QRS_NEXT_CUT()
PTP {E1 28976.891,E2 28976.891}
PTP {X 0,Y 607.92,A -85,B 0,C 180,E1 28976.891,E2 28976.891,E3 0,E4 0,E5 0,E6 0}
QRS_SPEED_INIT()
LIN {X 0,Y 607.92,Z 1028,A -85,B 0,C 180,E1 28976.891,E2 28976.891,E3 0,E4 0,E5 0,E6 0} C_VEL
LIN {X 0,Y 607.92,Z 449.836,A -85,B 0,C 180,E1 28976.891,E2 28976.891} C_VEL
LIN {X 0,Y 607.92,Z 441.762,A -85,B 0,C 180,E1 28976.891,E2 28976.891} C_VEL
LIN {X 0,Y 607.916,Z 439.762,A -85,B 0,C 180,E1 28976.702,E2 28976.702} C_VEL
LIN {X 0,Y 607.879,Z 439.765,A -85,B 0,C 180,E1 28973.483,E2 28973.483} C_VEL
LIN {X 0,Y 607.903,Z 439.761,A -85,B 0,C 180,E1 28970.246,E2 28970.246} C_VEL
LIN {X 0,Y 607.86,Z 439.764,A -85,B 0,C 180,E1 28967.266,E2 28967.266} C_VEL
LIN {X 0,Y 607.883,Z 439.762,A -85,B 0,C 180,E1 28963.959,E2 28963.959} C_VEL
LIN {X 0,Y 607.887,Z 439.761,A -85,B 0,C 180,E1 28960.894,E2 28960.894} C_VEL
LIN {X 0,Y 607.863,Z 439.765,A -85,B 0,C 180,E1 28957.668,E2 28957.668} C_VEL
LIN {X 0,Y 607.909,Z 439.763,A -85,B 0,C 180,E1 28954.682,E2 28954.682} C_VEL
LIN {X 0,Y 607.904,Z 439.766,A -85,B 0,C 180,E1 28951.511,E2 28951.511} C_VEL
LIN {X 0,Y 607.907,Z 439.765,A -85,B 0,C 180,E1 28948.353,E2 28948.353} C_VEL
LIN {X 0,Y 607.906,Z 439.763,A -85,B 0,C 180,E1 28945.158,E2 28945.158} C_VEL
LIN {X 0,Y 607.884,Z 439.763,A -85,B 0,C 180,E1 28942.036,E2 28942.036} C_VEL
LIN {X 0,Y 607.88,Z 439.763,A -85,B 0,C 180,E1 28938.857,E2 28938.857} C_VEL
LIN {X 0,Y 607.897,Z 439.76,A -85,B 0,C 180,E1 28935.782,E2 28935.782} C_VEL
LIN {X 0,Y 607.855,Z 439.765,A -85,B 0,C 180,E1 28932.535,E2 28932.535} C_VEL
LIN {X 0,Y 607.91,Z 439.76,A -85,B 0,C 180,E1 28929.521,E2 28929.521} C_VEL
LIN {X 0,Y 607.877,Z 439.765,A -85,B 0,C 180,E1 28926.296,E2 28926.296} C_VEL
LIN {X 0,Y 607.914,Z 439.762,A -85,B 0,C 180,E1 28923.096,E2 28923.096} C_VEL
LIN {X 0,Y 607.914,Z 439.902,A -85,B 0,C 180,E1 28921.609,E2 28921.609} C_VEL
LIN {X 0,Y 607.897,Z 481.904,A -85,B 0,C 180,E1 28918.56,E2 28918.56} C_VEL
LIN {X 0,Y 607.908,Z 495.16,A -85,B 0,C 180,E1 28917.629,E2 28917.629} C_VEL
LIN {X 0,Y 607.911,Z 733.402,A -85,B 0,C 180,E1 28914.557,E2 28914.557} C_VEL
LIN {X 0,Y 607.918,Z 759.72,A -85,B 0,C 180,E1 28914.175,E2 28914.175} C_VEL
LIN {X 0,Y 607.906,Z 779.969,A -85,B 0,C 180,E1 28913.712,E2 28913.712} C_VEL
LIN {X 0,Y 607.911,Z 800.64,A -85,B 0,C 180,E1 28913.044,E2 28913.044} C_VEL
LIN {X 0,Y 607.905,Z 820.106,A -85,B 0,C 180,E1 28912.228,E2 28912.228} C_VEL
LIN {X 0,Y 607.918,Z 838.721,A -85,B 0,C 180,E1 28911.263,E2 28911.263} C_VEL
LIN {X 0,Y 607.916,Z 857.259,A -85,B 0,C 180,E1 28910.105,E2 28910.105} C_VEL
LIN {X 0,Y 607.914,Z 874.073,A -85,B 0,C 180,E1 28908.855,E2 28908.855} C_VEL
LIN {X 0,Y 607.912,Z 890.09,A -85,B 0,C 180,E1 28907.455,E2 28907.455} C_VEL
LIN {X 0,Y 607.911,Z 904.816,A -85,B 0,C 180,E1 28905.942,E2 28905.942} C_VEL
LIN {X 0,Y 607.913,Z 918.531,A -85,B 0,C 180,E1 28904.282,E2 28904.282} C_VEL
LIN {X 0,Y 607.914,Z 930.639,A -85,B 0,C 180,E1 28902.539,E2 28902.539} C_VEL
LIN {X 0,Y 607.903,Z 940.638,A -85,B 0,C 180,E1 28900.807,E2 28900.807} C_VEL
LIN {X 0,Y 607.9,Z 949.278,A -85,B 0,C 180,E1 28898.989,E2 28898.989} C_VEL
LIN {X 0,Y 607.898,Z 956.152,A -85,B 0,C 180,E1 28897.18,E2 28897.18} C_VEL
LIN {X 0,Y 607.899,Z 961.632,A -85,B 0,C 180,E1 28895.284,E2 28895.284} C_VEL
LIN {X 0,Y 607.898,Z 965.323,A -85,B 0,C 180,E1 28893.394,E2 28893.394} C_VEL
LIN {X 0,Y 607.9,Z 967.407,A -85,B 0,C 180,E1 28891.507,E2 28891.507} C_VEL
LIN {X 0,Y 607.899,Z 967.906,A -85,B 0,C 180,E1 28889.528,E2 28889.528} C_VEL
LIN {X 0,Y 607.905,Z 966.779,A -85,B 0,C 180,E1 28887.643,E2 28887.643} C_VEL
LIN {X 0,Y 607.911,Z 963.877,A -85,B 0,C 180,E1 28885.66,E2 28885.66} C_VEL
LIN {X 0,Y 607.916,Z 959.347,A -85,B 0,C 180,E1 28883.768,E2 28883.768} C_VEL
LIN {X 0,Y 607.912,Z 953.368,A -85,B 0,C 180,E1 28881.946,E2 28881.946} C_VEL
LIN {X 0,Y 607.904,Z 945.39,A -85,B 0,C 180,E1 28880.055,E2 28880.055} C_VEL
LIN {X 0,Y 607.903,Z 936.41,A -85,B 0,C 180,E1 28878.328,E2 28878.328} C_VEL
LIN {X 0,Y 607.906,Z 925.469,A -85,B 0,C 180,E1 28876.59,E2 28876.59} C_VEL
LIN {X 0,Y 607.915,Z 913.063,A -85,B 0,C 180,E1 28874.937,E2 28874.937} C_VEL
LIN {X 0,Y 607.916,Z 899.235,A -85,B 0,C 180,E1 28873.37,E2 28873.37} C_VEL
LIN {X 0,Y 607.913,Z 883.891,A -85,B 0,C 180,E1 28871.889,E2 28871.889} C_VEL
LIN {X 0,Y 607.917,Z 867.529,A -85,B 0,C 180,E1 28870.545,E2 28870.545} C_VEL
LIN {X 0,Y 607.92,Z 850.05,A -85,B 0,C 180,E1 28869.329,E2 28869.329} C_VEL
LIN {X 0,Y 607.919,Z 832.125,A -85,B 0,C 180,E1 28868.28,E2 28868.28} C_VEL
LIN {X 0,Y 607.917,Z 813.106,A -85,B 0,C 180,E1 28867.364,E2 28867.364} C_VEL
LIN {X 0,Y 607.912,Z 794.381,A -85,B 0,C 180,E1 28866.647,E2 28866.647} C_VEL
LIN {X 0,Y 607.905,Z 774.324,A -85,B 0,C 180,E1 28866.055,E2 28866.055} C_VEL
LIN {X 0,Y 607.914,Z 754.612,A -85,B 0,C 180,E1 28865.643,E2 28865.643} C_VEL
LIN {X 0,Y 607.842,Z 497.544,A -85,B 0,C 180,E1 28862.309,E2 28862.309} C_VEL
LIN {X 0,Y 607.879,Z 470.838,A -85,B 0,C 180,E1 28859.452,E2 28859.452} C_VEL
LIN {X 0,Y 607.867,Z 443.132,A -85,B 0,C 180,E1 28856.393,E2 28856.393} C_VEL
LIN {X 0,Y 607.859,Z 439.766,A -85,B 0,C 180,E1 28855.995,E2 28855.995} C_VEL
LIN {X 0,Y 607.916,Z 439.759,A -85,B 0,C 180,E1 28852.87,E2 28852.87} C_VEL
LIN {X 0,Y 607.876,Z 439.762,A -85,B 0,C 180,E1 28849.748,E2 28849.748} C_VEL
LIN {X 0,Y 607.918,Z 439.755,A -85,B 0,C 180,E1 28846.567,E2 28846.567} C_VEL
LIN {X 0,Y 607.908,Z 439.765,A -85,B 0,C 180,E1 28843.304,E2 28843.304} C_VEL
LIN {X 0,Y 607.896,Z 439.757,A -85,B 0,C 180,E1 28840.024,E2 28840.024} C_VEL
LIN {X 0,Y 607.9,Z 439.762,A -85,B 0,C 180,E1 28836.895,E2 28836.895} C_VEL
LIN {X 0,Y 607.9,Z 439.758,A -85,B 0,C 180,E1 28833.775,E2 28833.775} C_VEL
LIN {X 0,Y 607.886,Z 439.761,A -85,B 0,C 180,E1 28830.656,E2 28830.656} C_VEL
LIN {X 0,Y 607.907,Z 439.761,A -85,B 0,C 180,E1 28827.528,E2 28827.528} C_VEL
LIN {X 0,Y 607.88,Z 439.77,A -85,B 0,C 180,E1 28826.547,E2 28826.547} C_VEL
LIN {X 0,Y 607.916,Z 471.412,A -85,B 0,C 180,E1 28823.712,E2 28823.712} C_VEL
LIN {X 0,Y 607.851,Z 506.361,A -85,B 0,C 180,E1 28820.711,E2 28820.711} C_VEL
LIN {X 0,Y 607.912,Z 542.01,A -85,B 0,C 180,E1 28817.715,E2 28817.715} C_VEL
LIN {X 0,Y 607.873,Z 578.969,A -85,B 0,C 180,E1 28814.673,E2 28814.673} C_VEL
LIN {X 0,Y 607.886,Z 602.408,A -85,B 0,C 180,E1 28812.779,E2 28812.779} C_VEL
LIN {X 0,Y 607.901,Z 743.315,A -85,B 0,C 180,E1 28811.071,E2 28811.071} C_VEL
LIN {X 0,Y 607.902,Z 760.125,A -85,B 0,C 180,E1 28810.687,E2 28810.687} C_VEL
LIN {X 0,Y 607.908,Z 774.888,A -85,B 0,C 180,E1 28810.184,E2 28810.184} C_VEL
LIN {X 0,Y 607.917,Z 789.399,A -85,B 0,C 180,E1 28809.515,E2 28809.515} C_VEL
LIN {X 0,Y 607.919,Z 804.496,A -85,B 0,C 180,E1 28808.608,E2 28808.608} C_VEL
LIN {X 0,Y 607.919,Z 817.563,A -85,B 0,C 180,E1 28807.608,E2 28807.608} C_VEL
LIN {X 0,Y 607.917,Z 829.982,A -85,B 0,C 180,E1 28806.422,E2 28806.422} C_VEL
LIN {X 0,Y 607.916,Z 840.212,A -85,B 0,C 180,E1 28805.19,E2 28805.19} C_VEL
LIN {X 0,Y 607.915,Z 849.003,A -85,B 0,C 180,E1 28803.867,E2 28803.867} C_VEL
LIN {X 0,Y 607.915,Z 856.257,A -85,B 0,C 180,E1 28802.451,E2 28802.451} C_VEL
LIN {X 0,Y 607.914,Z 861.91,A -85,B 0,C 180,E1 28800.943,E2 28800.943} C_VEL
LIN {X 0,Y 607.915,Z 865.679,A -85,B 0,C 180,E1 28799.435,E2 28799.435} C_VEL
LIN {X 0,Y 607.914,Z 867.614,A -85,B 0,C 180,E1 28797.926,E2 28797.926} C_VEL
LIN {X 0,Y 607.917,Z 867.88,A -85,B 0,C 180,E1 28796.417,E2 28796.417} C_VEL
LIN {X 0,Y 607.916,Z 866.393,A -85,B 0,C 180,E1 28794.905,E2 28794.905} C_VEL
LIN {X 0,Y 607.916,Z 863.141,A -85,B 0,C 180,E1 28793.389,E2 28793.389} C_VEL
LIN {X 0,Y 607.915,Z 858.333,A -85,B 0,C 180,E1 28791.947,E2 28791.947} C_VEL
LIN {X 0,Y 607.918,Z 851.731,A -85,B 0,C 180,E1 28790.534,E2 28790.534} C_VEL
LIN {X 0,Y 607.917,Z 843.602,A -85,B 0,C 180,E1 28789.193,E2 28789.193} C_VEL
LIN {X 0,Y 607.917,Z 834.031,A -85,B 0,C 180,E1 28787.943,E2 28787.943} C_VEL
LIN {X 0,Y 607.919,Z 822.43,A -85,B 0,C 180,E1 28786.736,E2 28786.736} C_VEL
LIN {X 0,Y 607.918,Z 810.297,A -85,B 0,C 180,E1 28785.717,E2 28785.717} C_VEL
LIN {X 0,Y 607.909,Z 796.446,A -85,B 0,C 180,E1 28784.791,E2 28784.791} C_VEL
LIN {X 0,Y 607.906,Z 782.578,A -85,B 0,C 180,E1 28784.058,E2 28784.058} C_VEL
LIN {X 0,Y 607.912,Z 767.197,A -85,B 0,C 180,E1 28783.444,E2 28783.444} C_VEL
LIN {X 0,Y 607.892,Z 751.424,A -85,B 0,C 180,E1 28783.001,E2 28783.001} C_VEL
LIN {X 0,Y 607.897,Z 734.775,A -85,B 0,C 180,E1 28782.717,E2 28782.717} C_VEL
LIN {X 0,Y 607.88,Z 602.145,A -85,B 0,C 180,E1 28781.118,E2 28781.118} C_VEL
LIN {X 0,Y 607.915,Z 563.557,A -85,B 0,C 180,E1 28777.976,E2 28777.976} C_VEL
LIN {X 0,Y 607.848,Z 527.624,A -85,B 0,C 180,E1 28774.992,E2 28774.992} C_VEL
LIN {X 0,Y 607.892,Z 490.334,A -85,B 0,C 180,E1 28771.832,E2 28771.832} C_VEL
LIN {X 0,Y 607.896,Z 466.16,A -85,B 0,C 180,E1 28769.714,E2 28769.714} C_VEL
LIN {X 0,Y 607.897,Z 441.985,A -85,B 0,C 180,E1 28767.073,E2 28767.073} C_VEL
LIN {X 0,Y 607.914,Z 439.765,A -85,B 0,C 180,E1 28766.791,E2 28766.791} C_VEL
LIN {X 0,Y 607.905,Z 439.758,A -85,B 0,C 180,E1 28763.542,E2 28763.542} C_VEL
LIN {X 0,Y 607.883,Z 439.762,A -85,B 0,C 180,E1 28760.465,E2 28760.465} C_VEL
LIN {X 0,Y 607.914,Z 439.762,A -85,B 0,C 180,E1 28757.325,E2 28757.325} C_VEL
LIN {X 0,Y 607.894,Z 439.92,A -85,B 0,C 180,E1 28754.948,E2 28754.948} C_VEL
LIN {X 0,Y 607.897,Z 476.657,A -85,B 0,C 180,E1 28752.789,E2 28752.789} C_VEL
LIN {X 0,Y 607.909,Z 521.292,A -85,B 0,C 180,E1 28750.256,E2 28750.256} C_VEL
LIN {X 0,Y 607.912,Z 533.861,A -85,B 0,C 180,E1 28749.374,E2 28749.374} C_VEL
LIN {X 0,Y 607.894,Z 542.903,A -85,B 0,C 180,E1 28748.564,E2 28748.564} C_VEL
LIN {X 0,Y 607.9,Z 548.563,A -85,B 0,C 180,E1 28747.844,E2 28747.844} C_VEL
LIN {X 0,Y 607.907,Z 550.683,A -85,B 0,C 180,E1 28747.367,E2 28747.367} C_VEL
LIN {X 0,Y 607.899,Z 550.949,A -85,B 0,C 180,E1 28746.931,E2 28746.931} C_VEL
LIN {X 0,Y 607.897,Z 549.412,A -85,B 0,C 180,E1 28746.616,E2 28746.616} C_VEL
LIN {X 0,Y 607.905,Z 546.003,A -85,B 0,C 180,E1 28746.366,E2 28746.366} C_VEL
LIN {X 0,Y 607.91,Z 540.136,A -85,B 0,C 180,E1 28746.191,E2 28746.191} C_VEL
LIN {X 0,Y 607.913,Z 532.275,A -85,B 0,C 180,E1 28746.13,E2 28746.13} C_VEL
LIN {X 0,Y 607.911,Z 439.764,A -85,B 0,C 180,E1 28746.108,E2 28746.108} C_VEL
LIN {X 0,Y 607.9,Z 439.909,A -85,B 0,C 180,E1 28743.988,E2 28743.988} C_VEL
LIN {X 0,Y 607.915,Z 489.526,A -85,B 0,C 180,E1 28740.93,E2 28740.93} C_VEL
LIN {X 0,Y 607.857,Z 537.557,A -85,B 0,C 180,E1 28738.063,E2 28738.063} C_VEL
LIN {X 0,Y 607.85,Z 544.1,A -85,B 0,C 180,E1 28737.691,E2 28737.691} C_VEL
LIN {X 0,Y 607.912,Z 784.325,A -85,B 0,C 180,E1 28734.59,E2 28734.59} C_VEL
LIN {X 0,Y 607.917,Z 810.634,A -85,B 0,C 180,E1 28734.202,E2 28734.202} C_VEL
LIN {X 0,Y 607.906,Z 830.575,A -85,B 0,C 180,E1 28733.739,E2 28733.739} C_VEL
LIN {X 0,Y 607.909,Z 851.165,A -85,B 0,C 180,E1 28733.071,E2 28733.071} C_VEL
LIN {X 0,Y 607.905,Z 871.073,A -85,B 0,C 180,E1 28732.229,E2 28732.229} C_VEL
LIN {X 0,Y 607.917,Z 889.502,A -85,B 0,C 180,E1 28731.264,E2 28731.264} C_VEL
LIN {X 0,Y 607.915,Z 908.095,A -85,B 0,C 180,E1 28730.092,E2 28730.092} C_VEL
LIN {X 0,Y 607.916,Z 925.213,A -85,B 0,C 180,E1 28728.807,E2 28728.807} C_VEL
LIN {X 0,Y 607.911,Z 940.921,A -85,B 0,C 180,E1 28727.419,E2 28727.419} C_VEL
LIN {X 0,Y 607.912,Z 955.198,A -85,B 0,C 180,E1 28725.943,E2 28725.943} C_VEL
LIN {X 0,Y 607.911,Z 968.852,A -85,B 0,C 180,E1 28724.284,E2 28724.284} C_VEL
LIN {X 0,Y 607.914,Z 980.927,A -85,B 0,C 180,E1 28722.54,E2 28722.54} C_VEL
LIN {X 0,Y 607.902,Z 991.394,A -85,B 0,C 180,E1 28720.712,E2 28720.712} C_VEL
LIN {X 0,Y 607.901,Z 999.872,A -85,B 0,C 180,E1 28718.895,E2 28718.895} C_VEL
LIN {X 0,Y 607.901,Z 1006.898,A -85,B 0,C 180,E1 28716.991,E2 28716.991} C_VEL
LIN {X 0,Y 607.901,Z 1012.142,A -85,B 0,C 180,E1 28715.096,E2 28715.096} C_VEL
LIN {X 0,Y 607.9,Z 1015.708,A -85,B 0,C 180,E1 28713.206,E2 28713.206} C_VEL
LIN {X 0,Y 607.9,Z 1017.572,A -85,B 0,C 180,E1 28711.32,E2 28711.32} C_VEL
LIN {X 0,Y 607.9,Z 1017.874,A -85,B 0,C 180,E1 28709.435,E2 28709.435} C_VEL
LIN {X 0,Y 607.906,Z 1016.504,A -85,B 0,C 180,E1 28707.455,E2 28707.455} C_VEL
LIN {X 0,Y 607.91,Z 1013.579,A -85,B 0,C 180,E1 28705.567,E2 28705.567} C_VEL
LIN {X 0,Y 607.916,Z 1008.976,A -85,B 0,C 180,E1 28703.674,E2 28703.674} C_VEL
LIN {X 0,Y 607.915,Z 1002.56,A -85,B 0,C 180,E1 28701.774,E2 28701.774} C_VEL
LIN {X 0,Y 607.904,Z 994.717,A -85,B 0,C 180,E1 28699.96,E2 28699.96} C_VEL
LIN {X 0,Y 607.906,Z 984.971,A -85,B 0,C 180,E1 28698.133,E2 28698.133} C_VEL
LIN {X 0,Y 607.914,Z 973.955,A -85,B 0,C 180,E1 28696.418,E2 28696.418} C_VEL
LIN {X 0,Y 607.912,Z 961.139,A -85,B 0,C 180,E1 28694.743,E2 28694.743} C_VEL
LIN {X 0,Y 607.913,Z 946.49,A -85,B 0,C 180,E1 28693.125,E2 28693.125} C_VEL
LIN {X 0,Y 607.917,Z 930.414,A -85,B 0,C 180,E1 28691.623,E2 28691.623} C_VEL
LIN {X 0,Y 607.919,Z 912.974,A -85,B 0,C 180,E1 28690.246,E2 28690.246} C_VEL
LIN {X 0,Y 607.919,Z 894.741,A -85,B 0,C 180,E1 28689.04,E2 28689.04} C_VEL
LIN {X 0,Y 607.91,Z 876.21,A -85,B 0,C 180,E1 28688.022,E2 28688.022} C_VEL
LIN {X 0,Y 607.913,Z 857.004,A -85,B 0,C 180,E1 28687.161,E2 28687.161} C_VEL
LIN {X 0,Y 607.912,Z 837.516,A -85,B 0,C 180,E1 28686.469,E2 28686.469} C_VEL
LIN {X 0,Y 607.909,Z 818.352,A -85,B 0,C 180,E1 28685.953,E2 28685.953} C_VEL
LIN {X 0,Y 607.913,Z 798.224,A -85,B 0,C 180,E1 28685.592,E2 28685.592} C_VEL
LIN {X 0,Y 607.851,Z 548.259,A -85,B 0,C 180,E1 28682.364,E2 28682.364} C_VEL
LIN {X 0,Y 607.849,Z 543.467,A -85,B 0,C 180,E1 28682.284,E2 28682.284} C_VEL
LIN {X 0,Y 607.915,Z 495.889,A -85,B 0,C 180,E1 28679.455,E2 28679.455} C_VEL
LIN {X 0,Y 607.892,Z 446.952,A -85,B 0,C 180,E1 28676.451,E2 28676.451} C_VEL
LIN {X 0,Y 607.902,Z 439.765,A -85,B 0,C 180,E1 28675.992,E2 28675.992} C_VEL
LIN {X 0,Y 607.913,Z 439.765,A -85,B 0,C 180,E1 28673.87,E2 28673.87} C_VEL
LIN {X 0,Y 607.912,Z 537.302,A -85,B 0,C 180,E1 28673.847,E2 28673.847} C_VEL
LIN {X 0,Y 607.907,Z 544.42,A -85,B 0,C 180,E1 28673.7,E2 28673.7} C_VEL
LIN {X 0,Y 607.899,Z 548.681,A -85,B 0,C 180,E1 28673.459,E2 28673.459} C_VEL
LIN {X 0,Y 607.896,Z 550.451,A -85,B 0,C 180,E1 28673.224,E2 28673.224} C_VEL
LIN {X 0,Y 607.91,Z 551.062,A -85,B 0,C 180,E1 28672.871,E2 28672.871} C_VEL
LIN {X 0,Y 607.9,Z 549.833,A -85,B 0,C 180,E1 28672.396,E2 28672.396} C_VEL
LIN {X 0,Y 607.919,Z 546.033,A -85,B 0,C 180,E1 28671.8,E2 28671.8} C_VEL
LIN {X 0,Y 607.894,Z 539.194,A -85,B 0,C 180,E1 28671.075,E2 28671.075} C_VEL
LIN {X 0,Y 607.903,Z 527.321,A -85,B 0,C 180,E1 28670.142,E2 28670.142} C_VEL
LIN {X 0,Y 607.906,Z 484.418,A -85,B 0,C 180,E1 28667.324,E2 28667.324} C_VEL
LIN {X 0,Y 607.914,Z 442.665,A -85,B 0,C 180,E1 28664.454,E2 28664.454} C_VEL
LIN {X 0,Y 607.886,Z 439.765,A -85,B 0,C 180,E1 28664.219,E2 28664.219} C_VEL
LIN {X 0,Y 607.91,Z 439.764,A -85,B 0,C 180,E1 28661.124,E2 28661.124} C_VEL
LIN {X 0,Y 607.909,Z 439.765,A -85,B 0,C 180,E1 28657.864,E2 28657.864} C_VEL
LIN {X 0,Y 607.918,Z 439.764,A -85,B 0,C 180,E1 28654.571,E2 28654.571} C_VEL
LIN {X 0,Y 607.912,Z 439.765,A -85,B 0,C 180,E1 28651.315,E2 28651.315} C_VEL
LIN {X 0,Y 607.895,Z 439.765,A -85,B 0,C 180,E1 28648.164,E2 28648.164} C_VEL
LIN {X 0,Y 607.893,Z 439.763,A -85,B 0,C 180,E1 28645.005,E2 28645.005} C_VEL
LIN {X 0,Y 607.909,Z 439.76,A -85,B 0,C 180,E1 28641.821,E2 28641.821} C_VEL
LIN {X 0,Y 607.864,Z 439.765,A -85,B 0,C 180,E1 28638.609,E2 28638.609} C_VEL
LIN {X 0,Y 607.916,Z 439.758,A -85,B 0,C 180,E1 28635.453,E2 28635.453} C_VEL
LIN {X 0,Y 607.857,Z 439.765,A -85,B 0,C 180,E1 28632.297,E2 28632.297} C_VEL
LIN {X 0,Y 607.899,Z 439.76,A -85,B 0,C 180,E1 28629.085,E2 28629.085} C_VEL
LIN {X 0,Y 607.886,Z 439.763,A -85,B 0,C 180,E1 28625.948,E2 28625.948} C_VEL
LIN {X 0,Y 607.884,Z 439.765,A -85,B 0,C 180,E1 28622.828,E2 28622.828} C_VEL
LIN {X 0,Y 607.913,Z 439.764,A -85,B 0,C 180,E1 28619.717,E2 28619.717} C_VEL
LIN {X 0,Y 607.916,Z 439.762,A -85,B 0,C 180,E1 28616.702,E2 28616.702} C_VEL
LIN {X 0,Y 606.91,Z 439.892,A -85,B 0,C 180,E1 28615.976,E2 28615.976} C_VEL
LIN {X 0,Y 600.441,Z 440.689,A -85,B 0,C 180,E1 28613.94,E2 28613.94} C_VEL
LIN {X 0,Y 599.947,Z 440.754,A -85,B 0,C 180,E1 28613.41,E2 28613.41} C_VEL
LIN {X 0,Y 599.965,Z 440.75,A -85,B 0,C 180,E1 28610.213,E2 28610.213} C_VEL
LIN {X 0,Y 599.925,Z 440.752,A -85,B 0,C 180,E1 28607.155,E2 28607.155} C_VEL
LIN {X 0,Y 599.944,Z 440.751,A -85,B 0,C 180,E1 28603.939,E2 28603.939} C_VEL
LIN {X 0,Y 599.95,Z 440.75,A -85,B 0,C 180,E1 28600.833,E2 28600.833} C_VEL
LIN {X 0,Y 599.918,Z 440.753,A -85,B 0,C 180,E1 28597.46,E2 28597.46} C_VEL
LIN {X 0,Y 599.97,Z 440.748,A -85,B 0,C 180,E1 28594.366,E2 28594.366} C_VEL
LIN {X 0,Y 599.931,Z 440.754,A -85,B 0,C 180,E1 28591.097,E2 28591.097} C_VEL
LIN {X 0,Y 599.974,Z 440.749,A -85,B 0,C 180,E1 28587.885,E2 28587.885} C_VEL
LIN {X 0,Y 599.958,Z 440.752,A -85,B 0,C 180,E1 28584.669,E2 28584.669} C_VEL
LIN {X 0,Y 599.97,Z 440.754,A -85,B 0,C 180,E1 28581.559,E2 28581.559} C_VEL
LIN {X 0,Y 599.979,Z 440.754,A -85,B 0,C 180,E1 28578.295,E2 28578.295} C_VEL
LIN {X 0,Y 599.975,Z 440.754,A -85,B 0,C 180,E1 28575.041,E2 28575.041} C_VEL
LIN {X 0,Y 599.958,Z 440.754,A -85,B 0,C 180,E1 28571.845,E2 28571.845} C_VEL
LIN {X 0,Y 599.963,Z 440.752,A -85,B 0,C 180,E1 28568.678,E2 28568.678} C_VEL
LIN {X 0,Y 599.941,Z 440.753,A -85,B 0,C 180,E1 28565.565,E2 28565.565} C_VEL
LIN {X 0,Y 599.939,Z 440.753,A -85,B 0,C 180,E1 28562.331,E2 28562.331} C_VEL
LIN {X 0,Y 599.975,Z 440.917,A -85,B 0,C 180,E1 28562.001,E2 28562.001} C_VEL
LIN {X 0,Y 600.713,Z 443.958,A -85,B 0,C 180,E1 28561.73,E2 28561.73} C_VEL
LIN {X 0,Y 600.551,Z 485.677,A -85,B 0,C 180,E1 28558.669,E2 28558.669} C_VEL
LIN {X 0,Y 600.626,Z 495.445,A -85,B 0,C 180,E1 28557.99,E2 28557.99} C_VEL
LIN {X 0,Y 600.675,Z 643.929,A -85,B 0,C 180,E1 28556.035,E2 28556.035} C_VEL
LIN {X 0,Y 600.615,Z 756.522,A -85,B 0,C 180,E1 28554.551,E2 28554.551} C_VEL
LIN {X 0,Y 600.558,Z 777.053,A -85,B 0,C 180,E1 28554.097,E2 28554.097} C_VEL
LIN {X 0,Y 600.499,Z 797.281,A -85,B 0,C 180,E1 28553.466,E2 28553.466} C_VEL
LIN {X 0,Y 600.42,Z 816.768,A -85,B 0,C 180,E1 28552.675,E2 28552.675} C_VEL
LIN {X 0,Y 600.347,Z 835.373,A -85,B 0,C 180,E1 28551.739,E2 28551.739} C_VEL
LIN {X 0,Y 600.277,Z 853.707,A -85,B 0,C 180,E1 28550.622,E2 28550.622} C_VEL
LIN {X 0,Y 600.195,Z 871.828,A -85,B 0,C 180,E1 28549.295,E2 28549.295} C_VEL
LIN {X 0,Y 600.123,Z 888.421,A -85,B 0,C 180,E1 28547.852,E2 28547.852} C_VEL
LIN {X 0,Y 600.058,Z 903.489,A -85,B 0,C 180,E1 28546.306,E2 28546.306} C_VEL
LIN {X 0,Y 600.01,Z 917.017,A -85,B 0,C 180,E1 28544.672,E2 28544.672} C_VEL
LIN {X 0,Y 599.971,Z 928.727,A -85,B 0,C 180,E1 28543.001,E2 28543.001} C_VEL
LIN {X 0,Y 599.943,Z 939.608,A -85,B 0,C 180,E1 28541.146,E2 28541.146} C_VEL
LIN {X 0,Y 599.924,Z 948.469,A -85,B 0,C 180,E1 28539.303,E2 28539.303} C_VEL
LIN {X 0,Y 599.915,Z 955.549,A -85,B 0,C 180,E1 28537.469,E2 28537.469} C_VEL
LIN {X 0,Y 599.91,Z 961.137,A -85,B 0,C 180,E1 28535.547,E2 28535.547} C_VEL
LIN {X 0,Y 599.907,Z 965.008,A -85,B 0,C 180,E1 28533.631,E2 28533.631} C_VEL
LIN {X 0,Y 599.904,Z 967.342,A -85,B 0,C 180,E1 28531.623,E2 28531.623} C_VEL
LIN {X 0,Y 599.904,Z 967.95,A -85,B 0,C 180,E1 28529.713,E2 28529.713} C_VEL
LIN {X 0,Y 599.912,Z 966.997,A -85,B 0,C 180,E1 28527.803,E2 28527.803} C_VEL
LIN {X 0,Y 599.916,Z 964.208,A -85,B 0,C 180,E1 28525.794,E2 28525.794} C_VEL
LIN {X 0,Y 599.918,Z 959.853,A -85,B 0,C 180,E1 28523.876,E2 28523.876} C_VEL
LIN {X 0,Y 599.922,Z 953.545,A -85,B 0,C 180,E1 28521.887,E2 28521.887} C_VEL
LIN {X 0,Y 599.925,Z 945.851,A -85,B 0,C 180,E1 28520.018,E2 28520.018} C_VEL
LIN {X 0,Y 599.946,Z 936.405,A -85,B 0,C 180,E1 28518.171,E2 28518.171} C_VEL
LIN {X 0,Y 599.977,Z 925.468,A -85,B 0,C 180,E1 28516.409,E2 28516.409} C_VEL
LIN {X 0,Y 600.018,Z 913.061,A -85,B 0,C 180,E1 28514.734,E2 28514.734} C_VEL
LIN {X 0,Y 600.069,Z 899.232,A -85,B 0,C 180,E1 28513.146,E2 28513.146} C_VEL
LIN {X 0,Y 600.136,Z 883.886,A -85,B 0,C 180,E1 28511.646,E2 28511.646} C_VEL
LIN {X 0,Y 600.208,Z 867.144,A -85,B 0,C 180,E1 28510.256,E2 28510.256} C_VEL
LIN {X 0,Y 600.292,Z 849.442,A -85,B 0,C 180,E1 28509.015,E2 28509.015} C_VEL
LIN {X 0,Y 600.375,Z 831.123,A -85,B 0,C 180,E1 28507.941,E2 28507.941} C_VEL
LIN {X 0,Y 600.45,Z 812.727,A -85,B 0,C 180,E1 28507.05,E2 28507.05} C_VEL
LIN {X 0,Y 600.507,Z 792.903,A -85,B 0,C 180,E1 28506.29,E2 28506.29} C_VEL
LIN {X 0,Y 600.565,Z 773.012,A -85,B 0,C 180,E1 28505.711,E2 28505.711} C_VEL
LIN {X 0,Y 600.621,Z 751.764,A -85,B 0,C 180,E1 28505.285,E2 28505.285} C_VEL
LIN {X 0,Y 600.752,Z 499.457,A -85,B 0,C 180,E1 28501.98,E2 28501.98} C_VEL
LIN {X 0,Y 600.291,Z 497.323,A -85,B 0,C 180,E1 28501.908,E2 28501.908} C_VEL
LIN {X 0,Y 600.471,Z 469.824,A -85,B 0,C 180,E1 28498.922,E2 28498.922} C_VEL
LIN {X 0,Y 600.513,Z 442.981,A -85,B 0,C 180,E1 28495.909,E2 28495.909} C_VEL
LIN {X 0,Y 599.942,Z 440.757,A -85,B 0,C 180,E1 28495.585,E2 28495.585} C_VEL
LIN {X 0,Y 599.937,Z 440.749,A -85,B 0,C 180,E1 28492.291,E2 28492.291} C_VEL
LIN {X 0,Y 599.976,Z 440.753,A -85,B 0,C 180,E1 28489.165,E2 28489.165} C_VEL
LIN {X 0,Y 599.941,Z 440.748,A -85,B 0,C 180,E1 28485.974,E2 28485.974} C_VEL
LIN {X 0,Y 599.966,Z 440.749,A -85,B 0,C 180,E1 28482.838,E2 28482.838} C_VEL
LIN {X 0,Y 599.954,Z 440.75,A -85,B 0,C 180,E1 28479.65,E2 28479.65} C_VEL
LIN {X 0,Y 599.962,Z 440.747,A -85,B 0,C 180,E1 28476.51,E2 28476.51} C_VEL
LIN {X 0,Y 599.976,Z 440.755,A -85,B 0,C 180,E1 28473.218,E2 28473.218} C_VEL
LIN {X 0,Y 599.973,Z 440.746,A -85,B 0,C 180,E1 28469.887,E2 28469.887} C_VEL
LIN {X 0,Y 599.982,Z 440.948,A -85,B 0,C 180,E1 28466.901,E2 28466.901} C_VEL
LIN {X 0,Y 600.562,Z 444.397,A -85,B 0,C 180,E1 28466.553,E2 28466.553} C_VEL
LIN {X 0,Y 600.46,Z 473.908,A -85,B 0,C 180,E1 28463.868,E2 28463.868} C_VEL
LIN {X 0,Y 600.249,Z 508.414,A -85,B 0,C 180,E1 28460.854,E2 28460.854} C_VEL
LIN {X 0,Y 600.222,Z 544.422,A -85,B 0,C 180,E1 28457.79,E2 28457.79} C_VEL
LIN {X 0,Y 600.1,Z 581.875,A -85,B 0,C 180,E1 28454.67,E2 28454.67} C_VEL
LIN {X 0,Y 600.109,Z 602.615,A -85,B 0,C 180,E1 28452.987,E2 28452.987} C_VEL
LIN {X 0,Y 600.137,Z 744.248,A -85,B 0,C 180,E1 28451.241,E2 28451.241} C_VEL
LIN {X 0,Y 600.116,Z 761.589,A -85,B 0,C 180,E1 28450.828,E2 28450.828} C_VEL
LIN {X 0,Y 600.084,Z 777.042,A -85,B 0,C 180,E1 28450.27,E2 28450.27} C_VEL
LIN {X 0,Y 600.062,Z 792.809,A -85,B 0,C 180,E1 28449.495,E2 28449.495} C_VEL
LIN {X 0,Y 600.024,Z 806.446,A -85,B 0,C 180,E1 28448.626,E2 28448.626} C_VEL
LIN {X 0,Y 599.992,Z 819.677,A -85,B 0,C 180,E1 28447.565,E2 28447.565} C_VEL
LIN {X 0,Y 599.962,Z 831.185,A -85,B 0,C 180,E1 28446.411,E2 28446.411} C_VEL
LIN {X 0,Y 599.942,Z 841.21,A -85,B 0,C 180,E1 28445.164,E2 28445.164} C_VEL
LIN {X 0,Y 599.927,Z 849.793,A -85,B 0,C 180,E1 28443.823,E2 28443.823} C_VEL
LIN {X 0,Y 599.919,Z 856.828,A -85,B 0,C 180,E1 28442.388,E2 28442.388} C_VEL
LIN {X 0,Y 599.916,Z 862.34,A -85,B 0,C 180,E1 28440.86,E2 28440.86} C_VEL
LIN {X 0,Y 599.914,Z 865.897,A -85,B 0,C 180,E1 28439.332,E2 28439.332} C_VEL
LIN {X 0,Y 599.912,Z 867.773,A -85,B 0,C 180,E1 28437.708,E2 28437.708} C_VEL
LIN {X 0,Y 599.913,Z 867.756,A -85,B 0,C 180,E1 28436.178,E2 28436.178} C_VEL
LIN {X 0,Y 599.915,Z 866.005,A -85,B 0,C 180,E1 28434.645,E2 28434.645} C_VEL
LIN {X 0,Y 599.915,Z 862.516,A -85,B 0,C 180,E1 28433.108,E2 28433.108} C_VEL
LIN {X 0,Y 599.919,Z 857.016,A -85,B 0,C 180,E1 28431.566,E2 28431.566} C_VEL
LIN {X 0,Y 599.927,Z 849.944,A -85,B 0,C 180,E1 28430.116,E2 28430.116} C_VEL
LIN {X 0,Y 599.944,Z 841.279,A -85,B 0,C 180,E1 28428.756,E2 28428.756} C_VEL
LIN {X 0,Y 599.961,Z 831.088,A -85,B 0,C 180,E1 28427.488,E2 28427.488} C_VEL
LIN {X 0,Y 599.993,Z 819.862,A -85,B 0,C 180,E1 28426.361,E2 28426.361} C_VEL
LIN {X 0,Y 600.022,Z 807.05,A -85,B 0,C 180,E1 28425.328,E2 28425.328} C_VEL
LIN {X 0,Y 600.059,Z 793.245,A -85,B 0,C 180,E1 28424.439,E2 28424.439} C_VEL
LIN {X 0,Y 600.084,Z 777.161,A -85,B 0,C 180,E1 28423.645,E2 28423.645} C_VEL
LIN {X 0,Y 600.109,Z 762.099,A -85,B 0,C 180,E1 28423.098,E2 28423.098} C_VEL
LIN {X 0,Y 600.129,Z 744.807,A -85,B 0,C 180,E1 28422.68,E2 28422.68} C_VEL
LIN {X 0,Y 600.173,Z 692.301,A -85,B 0,C 180,E1 28422.015,E2 28422.015} C_VEL
LIN {X 0,Y 600.062,Z 602.228,A -85,B 0,C 180,E1 28420.913,E2 28420.913} C_VEL
LIN {X 0,Y 600.161,Z 563.636,A -85,B 0,C 180,E1 28417.728,E2 28417.728} C_VEL
LIN {X 0,Y 600.196,Z 528.321,A -85,B 0,C 180,E1 28414.757,E2 28414.757} C_VEL
LIN {X 0,Y 600.331,Z 490.404,A -85,B 0,C 180,E1 28411.499,E2 28411.499} C_VEL
LIN {X 0,Y 601.314,Z 468.18,A -85,B 0,C 180,E1 28409.28,E2 28409.28} C_VEL
LIN {X 0,Y 601.56,Z 444.633,A -85,B 0,C 180,E1 28406.651,E2 28406.651} C_VEL
LIN {X 0,Y 600.068,Z 441.359,A -85,B 0,C 180,E1 28406.069,E2 28406.069} C_VEL
LIN {X 0,Y 599.977,Z 440.748,A -85,B 0,C 180,E1 28405.92,E2 28405.92} C_VEL
LIN {X 0,Y 599.96,Z 440.754,A -85,B 0,C 180,E1 28402.651,E2 28402.651} C_VEL
LIN {X 0,Y 599.973,Z 440.75,A -85,B 0,C 180,E1 28399.458,E2 28399.458} C_VEL
LIN {X 0,Y 599.924,Z 440.754,A -85,B 0,C 180,E1 28396.33,E2 28396.33} C_VEL
LIN {X 0,Y 599.997,Z 440.89,A -85,B 0,C 180,E1 28395.447,E2 28395.447} C_VEL
LIN {X 0,Y 600.994,Z 444.439,A -85,B 0,C 180,E1 28395.132,E2 28395.132} C_VEL
LIN {X 0,Y 600.644,Z 478.663,A -85,B 0,C 180,E1 28393.048,E2 28393.048} C_VEL
LIN {X 0,Y 601.025,Z 532.786,A -85,B 0,C 180,E1 28389.953,E2 28389.953} C_VEL
LIN {X 0,Y 602.055,Z 544.781,A -85,B 0,C 180,E1 28389.131,E2 28389.131} C_VEL
LIN {X 0,Y 603.137,Z 552.148,A -85,B 0,C 180,E1 28388.438,E2 28388.438} C_VEL
LIN {X 0,Y 604.076,Z 556.322,A -85,B 0,C 180,E1 28387.859,E2 28387.859} C_VEL
LIN {X 0,Y 604.889,Z 558.286,A -85,B 0,C 180,E1 28387.338,E2 28387.338} C_VEL
LIN {X 0,Y 605.442,Z 558.491,A -85,B 0,C 180,E1 28386.833,E2 28386.833} C_VEL
LIN {X 0,Y 605.59,Z 556.888,A -85,B 0,C 180,E1 28386.381,E2 28386.381} C_VEL
LIN {X 0,Y 605.276,Z 553.74,A -85,B 0,C 180,E1 28386.011,E2 28386.011} C_VEL
LIN {X 0,Y 604.557,Z 548.711,A -85,B 0,C 180,E1 28385.727,E2 28385.727} C_VEL
LIN {X 0,Y 603.605,Z 541.502,A -85,B 0,C 180,E1 28385.566,E2 28385.566} C_VEL
LIN {X 0,Y 603.233,Z 532.842,A -85,B 0,C 180,E1 28385.516,E2 28385.516} C_VEL
LIN {X 0,Y 603.096,Z 446.156,A -85,B 0,C 180,E1 28385.498,E2 28385.498} C_VEL
LIN {X 0,Y 600.855,Z 443.524,A -85,B 0,C 180,E1 28385.198,E2 28385.198} C_VEL
LIN {X 0,Y 599.972,Z 440.745,A -85,B 0,C 180,E1 28385.061,E2 28385.061} C_VEL
LIN {X 0,Y 599.974,Z 440.808,A -85,B 0,C 180,E1 28384.443,E2 28384.443} C_VEL
LIN {X 0,Y 600.92,Z 444.123,A -85,B 0,C 180,E1 28384.17,E2 28384.17} C_VEL
LIN {X 0,Y 600.771,Z 493.151,A -85,B 0,C 180,E1 28381.116,E2 28381.116} C_VEL
LIN {X 0,Y 600.564,Z 541.182,A -85,B 0,C 180,E1 28378.218,E2 28378.218} C_VEL
LIN {X 0,Y 600.67,Z 544.583,A -85,B 0,C 180,E1 28378.044,E2 28378.044} C_VEL
LIN {X 0,Y 600.645,Z 723.632,A -85,B 0,C 180,E1 28375.694,E2 28375.694} C_VEL
LIN {X 0,Y 600.613,Z 806.807,A -85,B 0,C 180,E1 28374.591,E2 28374.591} C_VEL
LIN {X 0,Y 600.557,Z 827.719,A -85,B 0,C 180,E1 28374.126,E2 28374.126} C_VEL
LIN {X 0,Y 600.498,Z 847.519,A -85,B 0,C 180,E1 28373.502,E2 28373.502} C_VEL
LIN {X 0,Y 600.418,Z 867.263,A -85,B 0,C 180,E1 28372.697,E2 28372.697} C_VEL
LIN {X 0,Y 600.346,Z 886.153,A -85,B 0,C 180,E1 28371.739,E2 28371.739} C_VEL
LIN {X 0,Y 600.265,Z 904.337,A -85,B 0,C 180,E1 28370.623,E2 28370.623} C_VEL
LIN {X 0,Y 600.196,Z 921.557,A -85,B 0,C 180,E1 28369.361,E2 28369.361} C_VEL
LIN {X 0,Y 600.122,Z 938.362,A -85,B 0,C 180,E1 28367.903,E2 28367.903} C_VEL
LIN {X 0,Y 600.056,Z 953.438,A -85,B 0,C 180,E1 28366.356,E2 28366.356} C_VEL
LIN {X 0,Y 600.01,Z 967.365,A -85,B 0,C 180,E1 28364.673,E2 28364.673} C_VEL
LIN {X 0,Y 599.973,Z 979.011,A -85,B 0,C 180,E1 28363.002,E2 28363.002} C_VEL
LIN {X 0,Y 599.946,Z 989.324,A -85,B 0,C 180,E1 28361.245,E2 28361.245} C_VEL
LIN {X 0,Y 599.925,Z 998.365,A -85,B 0,C 180,E1 28359.373,E2 28359.373} C_VEL
LIN {X 0,Y 599.913,Z 1005.686,A -85,B 0,C 180,E1 28357.47,E2 28357.47} C_VEL
LIN {X 0,Y 599.907,Z 1011.252,A -85,B 0,C 180,E1 28355.548,E2 28355.548} C_VEL
LIN {X 0,Y 599.906,Z 1015.085,A -85,B 0,C 180,E1 28353.632,E2 28353.632} C_VEL
LIN {X 0,Y 599.902,Z 1017.375,A -85,B 0,C 180,E1 28351.624,E2 28351.624} C_VEL
LIN {X 0,Y 599.9,Z 1017.918,A -85,B 0,C 180,E1 28349.619,E2 28349.619} C_VEL
LIN {X 0,Y 599.908,Z 1016.843,A -85,B 0,C 180,E1 28347.708,E2 28347.708} C_VEL
LIN {X 0,Y 599.913,Z 1013.974,A -85,B 0,C 180,E1 28345.699,E2 28345.699} C_VEL
LIN {X 0,Y 599.919,Z 1009.481,A -85,B 0,C 180,E1 28343.781,E2 28343.781} C_VEL
LIN {X 0,Y 599.923,Z 1003.271,A -85,B 0,C 180,E1 28341.856,E2 28341.856} C_VEL
LIN {X 0,Y 599.926,Z 995.182,A -85,B 0,C 180,E1 28339.922,E2 28339.922} C_VEL
LIN {X 0,Y 599.949,Z 985.565,A -85,B 0,C 180,E1 28338.074,E2 28338.074} C_VEL
LIN {X 0,Y 599.989,Z 974.416,A -85,B 0,C 180,E1 28336.299,E2 28336.299} C_VEL
LIN {X 0,Y 600.027,Z 961.132,A -85,B 0,C 180,E1 28334.537,E2 28334.537} C_VEL
LIN {X 0,Y 600.09,Z 946.49,A -85,B 0,C 180,E1 28332.898,E2 28332.898} C_VEL
LIN {X 0,Y 600.15,Z 931.058,A -85,B 0,C 180,E1 28331.434,E2 28331.434} C_VEL
LIN {X 0,Y 600.221,Z 914.316,A -85,B 0,C 180,E1 28330.083,E2 28330.083} C_VEL
LIN {X 0,Y 600.298,Z 897.155,A -85,B 0,C 180,E1 28328.914,E2 28328.914} C_VEL
LIN {X 0,Y 600.377,Z 879.288,A -85,B 0,C 180,E1 28327.891,E2 28327.891} C_VEL
LIN {X 0,Y 600.458,Z 860.819,A -85,B 0,C 180,E1 28327.015,E2 28327.015} C_VEL
LIN {X 0,Y 600.516,Z 841.214,A -85,B 0,C 180,E1 28326.276,E2 28326.276} C_VEL
LIN {X 0,Y 600.569,Z 821.146,A -85,B 0,C 180,E1 28325.709,E2 28325.709} C_VEL
LIN {X 0,Y 600.621,Z 800.654,A -85,B 0,C 180,E1 28325.313,E2 28325.313} C_VEL
LIN {X 0,Y 600.761,Z 547.279,A -85,B 0,C 180,E1 28321.996,E2 28321.996} C_VEL
LIN {X 0,Y 600.553,Z 543.713,A -85,B 0,C 180,E1 28321.932,E2 28321.932} C_VEL
LIN {X 0,Y 600.762,Z 495.889,A -85,B 0,C 180,E1 28319.052,E2 28319.052} C_VEL
LIN {X 0,Y 600.903,Z 447.858,A -85,B 0,C 180,E1 28316.066,E2 28316.066} C_VEL
LIN {X 0,Y 600.75,Z 443.327,A -85,B 0,C 180,E1 28315.768,E2 28315.768} C_VEL
LIN {X 0,Y 599.966,Z 440.753,A -85,B 0,C 180,E1 28315.544,E2 28315.544} C_VEL
LIN {X 0,Y 599.994,Z 440.902,A -85,B 0,C 180,E1 28314.919,E2 28314.919} C_VEL
LIN {X 0,Y 601.065,Z 443.896,A -85,B 0,C 180,E1 28314.774,E2 28314.774} C_VEL
LIN {X 0,Y 603.229,Z 446.254,A -85,B 0,C 180,E1 28314.484,E2 28314.484} C_VEL
LIN {X 0,Y 603.381,Z 538.286,A -85,B 0,C 180,E1 28314.464,E2 28314.464} C_VEL
LIN {X 0,Y 604.264,Z 546.719,A -85,B 0,C 180,E1 28314.337,E2 28314.337} C_VEL
LIN {X 0,Y 605.074,Z 552.238,A -85,B 0,C 180,E1 28314.098,E2 28314.098} C_VEL
LIN {X 0,Y 605.534,Z 556.108,A -85,B 0,C 180,E1 28313.742,E2 28313.742} C_VEL
LIN {X 0,Y 605.563,Z 558.021,A -85,B 0,C 180,E1 28313.364,E2 28313.364} C_VEL
LIN {X 0,Y 605.207,Z 558.61,A -85,B 0,C 180,E1 28312.915,E2 28312.915} C_VEL
LIN {X 0,Y 604.477,Z 557.451,A -85,B 0,C 180,E1 28312.385,E2 28312.385} C_VEL
LIN {X 0,Y 603.576,Z 554.393,A -85,B 0,C 180,E1 28311.838,E2 28311.838} C_VEL
LIN {X 0,Y 602.422,Z 547.69,A -85,B 0,C 180,E1 28311.115,E2 28311.115} C_VEL
LIN {X 0,Y 601.39,Z 537.283,A -85,B 0,C 180,E1 28310.326,E2 28310.326} C_VEL
LIN {X 0,Y 601.231,Z 486.365,A -85,B 0,C 180,E1 28306.942,E2 28306.942} C_VEL
LIN {X 0,Y 601.438,Z 444.929,A -85,B 0,C 180,E1 28304.058,E2 28304.058} C_VEL
LIN {X 0,Y 599.925,Z 440.756,A -85,B 0,C 180,E1 28303.612,E2 28303.612} C_VEL
LIN {X 0,Y 599.976,Z 440.748,A -85,B 0,C 180,E1 28300.411,E2 28300.411} C_VEL
LIN {X 0,Y 599.918,Z 440.754,A -85,B 0,C 180,E1 28297.188,E2 28297.188} C_VEL
LIN {X 0,Y 599.963,Z 440.749,A -85,B 0,C 180,E1 28293.937,E2 28293.937} C_VEL
LIN {X 0,Y 599.943,Z 440.752,A -85,B 0,C 180,E1 28290.773,E2 28290.773} C_VEL
LIN {X 0,Y 599.938,Z 440.753,A -85,B 0,C 180,E1 28287.548,E2 28287.548} C_VEL
LIN {X 0,Y 599.967,Z 440.752,A -85,B 0,C 180,E1 28284.412,E2 28284.412} C_VEL
LIN {X 0,Y 599.96,Z 440.754,A -85,B 0,C 180,E1 28281.201,E2 28281.201} C_VEL
LIN {X 0,Y 599.977,Z 440.752,A -85,B 0,C 180,E1 28277.907,E2 28277.907} C_VEL
LIN {X 0,Y 599.973,Z 440.754,A -85,B 0,C 180,E1 28274.673,E2 28274.673} C_VEL
LIN {X 0,Y 599.972,Z 440.754,A -85,B 0,C 180,E1 28271.438,E2 28271.438} C_VEL
LIN {X 0,Y 599.973,Z 440.754,A -85,B 0,C 180,E1 28268.143,E2 28268.143} C_VEL
LIN {X 0,Y 599.977,Z 440.752,A -85,B 0,C 180,E1 28264.875,E2 28264.875} C_VEL
LIN {X 0,Y 599.957,Z 440.754,A -85,B 0,C 180,E1 28261.623,E2 28261.623} C_VEL
LIN {X 0,Y 599.968,Z 440.751,A -85,B 0,C 180,E1 28258.376,E2 28258.376} C_VEL
LIN {X 0,Y 599.928,Z 440.754,A -85,B 0,C 180,E1 28255.299,E2 28255.299} C_VEL
LIN {X 0,Y 599.947,Z 440.754,A -85,B 0,C 180,E1 28253.41,E2 28253.41} C_VEL
LIN {X 0,Y 599.007,Z 440.875,A -85,B 0,C 180,E1 28252.674,E2 28252.674} C_VEL
LIN {X 0,Y 592.559,Z 441.671,A -85,B 0,C 180,E1 28250.61,E2 28250.61} C_VEL
LIN {X 0,Y 592.029,Z 441.74,A -85,B 0,C 180,E1 28250.073,E2 28250.073} C_VEL
LIN {X 0,Y 591.999,Z 441.741,A -85,B 0,C 180,E1 28246.919,E2 28246.919} C_VEL
LIN {X 0,Y 592.006,Z 441.741,A -85,B 0,C 180,E1 28243.718,E2 28243.718} C_VEL
LIN {X 0,Y 592.022,Z 441.737,A -85,B 0,C 180,E1 28240.566,E2 28240.566} C_VEL
LIN {X 0,Y 591.979,Z 441.741,A -85,B 0,C 180,E1 28237.35,E2 28237.35} C_VEL
LIN {X 0,Y 592.037,Z 441.735,A -85,B 0,C 180,E1 28234.169,E2 28234.169} C_VEL
LIN {X 0,Y 591.988,Z 441.743,A -85,B 0,C 180,E1 28231.004,E2 28231.004} C_VEL
LIN {X 0,Y 592.023,Z 441.739,A -85,B 0,C 180,E1 28227.745,E2 28227.745} C_VEL
LIN {X 0,Y 592.017,Z 441.741,A -85,B 0,C 180,E1 28224.599,E2 28224.599} C_VEL
LIN {X 0,Y 592.016,Z 441.743,A -85,B 0,C 180,E1 28221.44,E2 28221.44} C_VEL
LIN {X 0,Y 592.04,Z 441.742,A -85,B 0,C 180,E1 28218.284,E2 28218.284} C_VEL
LIN {X 0,Y 592.032,Z 441.743,A -85,B 0,C 180,E1 28214.957,E2 28214.957} C_VEL
LIN {X 0,Y 592.035,Z 441.743,A -85,B 0,C 180,E1 28211.713,E2 28211.713} C_VEL
LIN {X 0,Y 592.033,Z 441.743,A -85,B 0,C 180,E1 28208.406,E2 28208.406} C_VEL
LIN {X 0,Y 592.035,Z 441.743,A -85,B 0,C 180,E1 28205.162,E2 28205.162} C_VEL
LIN {X 0,Y 592.018,Z 441.885,A -85,B 0,C 180,E1 28202.411,E2 28202.411} C_VEL
LIN {X 0,Y 593.521,Z 446.926,A -85,B 0,C 180,E1 28201.935,E2 28201.935} C_VEL
LIN {X 0,Y 593.218,Z 488.177,A -85,B 0,C 180,E1 28198.874,E2 28198.874} C_VEL
LIN {X 0,Y 593.27,Z 495.434,A -85,B 0,C 180,E1 28198.369,E2 28198.369} C_VEL
LIN {X 0,Y 593.75,Z 499.897,A -85,B 0,C 180,E1 28198.284,E2 28198.284} C_VEL
LIN {X 0,Y 593.369,Z 740.009,A -85,B 0,C 180,E1 28195.115,E2 28195.115} C_VEL
LIN {X 0,Y 593.304,Z 763.049,A -85,B 0,C 180,E1 28194.744,E2 28194.744} C_VEL
LIN {X 0,Y 593.179,Z 783.776,A -85,B 0,C 180,E1 28194.223,E2 28194.223} C_VEL
LIN {X 0,Y 593.053,Z 803.375,A -85,B 0,C 180,E1 28193.551,E2 28193.551} C_VEL
LIN {X 0,Y 592.904,Z 823.443,A -85,B 0,C 180,E1 28192.664,E2 28192.664} C_VEL
LIN {X 0,Y 592.754,Z 842.212,A -85,B 0,C 180,E1 28191.632,E2 28191.632} C_VEL
LIN {X 0,Y 592.588,Z 859.46,A -85,B 0,C 180,E1 28190.494,E2 28190.494} C_VEL
LIN {X 0,Y 592.429,Z 876.505,A -85,B 0,C 180,E1 28189.163,E2 28189.163} C_VEL
LIN {X 0,Y 592.286,Z 892.806,A -85,B 0,C 180,E1 28187.66,E2 28187.66} C_VEL
LIN {X 0,Y 592.171,Z 907.379,A -85,B 0,C 180,E1 28186.075,E2 28186.075} C_VEL
LIN {X 0,Y 592.078,Z 920.665,A -85,B 0,C 180,E1 28184.373,E2 28184.373} C_VEL
LIN {X 0,Y 592.019,Z 931.847,A -85,B 0,C 180,E1 28182.682,E2 28182.682} C_VEL
LIN {X 0,Y 591.963,Z 942.189,A -85,B 0,C 180,E1 28180.806,E2 28180.806} C_VEL
LIN {X 0,Y 591.929,Z 950.505,A -85,B 0,C 180,E1 28178.94,E2 28178.94} C_VEL
LIN {X 0,Y 591.909,Z 957.066,A -85,B 0,C 180,E1 28177.083,E2 28177.083} C_VEL
LIN {X 0,Y 591.904,Z 962.254,A -85,B 0,C 180,E1 28175.136,E2 28175.136} C_VEL
LIN {X 0,Y 591.899,Z 965.779,A -85,B 0,C 180,E1 28173.195,E2 28173.195} C_VEL
LIN {X 0,Y 591.9,Z 967.608,A -85,B 0,C 180,E1 28171.258,E2 28171.258} C_VEL
LIN {X 0,Y 591.902,Z 967.862,A -85,B 0,C 180,E1 28169.322,E2 28169.322} C_VEL
LIN {X 0,Y 591.908,Z 966.443,A -85,B 0,C 180,E1 28167.288,E2 28167.288} C_VEL
LIN {X 0,Y 591.915,Z 963.349,A -85,B 0,C 180,E1 28165.293,E2 28165.293} C_VEL
LIN {X 0,Y 591.925,Z 958.55,A -85,B 0,C 180,E1 28163.306,E2 28163.306} C_VEL
LIN {X 0,Y 591.936,Z 952.013,A -85,B 0,C 180,E1 28161.353,E2 28161.353} C_VEL
LIN {X 0,Y 591.962,Z 944.004,A -85,B 0,C 180,E1 28159.489,E2 28159.489} C_VEL
LIN {X 0,Y 592.009,Z 934.097,A -85,B 0,C 180,E1 28157.614,E2 28157.614} C_VEL
LIN {X 0,Y 592.066,Z 922.706,A -85,B 0,C 180,E1 28155.825,E2 28155.825} C_VEL
LIN {X 0,Y 592.161,Z 909.827,A -85,B 0,C 180,E1 28154.125,E2 28154.125} C_VEL
LIN {X 0,Y 592.276,Z 895.418,A -85,B 0,C 180,E1 28152.512,E2 28152.512} C_VEL
LIN {X 0,Y 592.416,Z 879.957,A -85,B 0,C 180,E1 28151.04,E2 28151.04} C_VEL
LIN {X 0,Y 592.567,Z 862.874,A -85,B 0,C 180,E1 28149.659,E2 28149.659} C_VEL
LIN {X 0,Y 592.726,Z 844.616,A -85,B 0,C 180,E1 28148.423,E2 28148.423} C_VEL
LIN {X 0,Y 592.861,Z 826.143,A -85,B 0,C 180,E1 28147.385,E2 28147.385} C_VEL
LIN {X 0,Y 593.025,Z 807.309,A -85,B 0,C 180,E1 28146.521,E2 28146.521} C_VEL
LIN {X 0,Y 593.173,Z 786.971,A -85,B 0,C 180,E1 28145.784,E2 28145.784} C_VEL
LIN {X 0,Y 593.286,Z 766.686,A -85,B 0,C 180,E1 28145.241,E2 28145.241} C_VEL
LIN {X 0,Y 593.362,Z 745.735,A -85,B 0,C 180,E1 28144.87,E2 28144.87} C_VEL
LIN {X 0,Y 593.681,Z 501.052,A -85,B 0,C 180,E1 28141.638,E2 28141.638} C_VEL
LIN {X 0,Y 592.768,Z 497.387,A -85,B 0,C 180,E1 28141.526,E2 28141.526} C_VEL
LIN {X 0,Y 593.023,Z 468.809,A -85,B 0,C 180,E1 28138.374,E2 28138.374} C_VEL
LIN {X 0,Y 593.144,Z 445.884,A -85,B 0,C 180,E1 28135.764,E2 28135.764} C_VEL
LIN {X 0,Y 592.034,Z 441.743,A -85,B 0,C 180,E1 28135.191,E2 28135.191} C_VEL
LIN {X 0,Y 591.991,Z 441.74,A -85,B 0,C 180,E1 28132.063,E2 28132.063} C_VEL
LIN {X 0,Y 592.035,Z 441.739,A -85,B 0,C 180,E1 28128.931,E2 28128.931} C_VEL
LIN {X 0,Y 592.003,Z 441.739,A -85,B 0,C 180,E1 28125.735,E2 28125.735} C_VEL
LIN {X 0,Y 592.033,Z 441.734,A -85,B 0,C 180,E1 28122.497,E2 28122.497} C_VEL
LIN {X 0,Y 592.036,Z 441.743,A -85,B 0,C 180,E1 28119.171,E2 28119.171} C_VEL
LIN {X 0,Y 592.022,Z 441.737,A -85,B 0,C 180,E1 28115.838,E2 28115.838} C_VEL
LIN {X 0,Y 592.014,Z 441.741,A -85,B 0,C 180,E1 28112.715,E2 28112.715} C_VEL
LIN {X 0,Y 592.027,Z 441.741,A -85,B 0,C 180,E1 28109.548,E2 28109.548} C_VEL
LIN {X 0,Y 592.06,Z 441.918,A -85,B 0,C 180,E1 28107.291,E2 28107.291} C_VEL
LIN {X 0,Y 593.253,Z 447.025,A -85,B 0,C 180,E1 28106.744,E2 28106.744} C_VEL
LIN {X 0,Y 593.069,Z 477.32,A -85,B 0,C 180,E1 28103.968,E2 28103.968} C_VEL
LIN {X 0,Y 592.65,Z 510.375,A -85,B 0,C 180,E1 28101.009,E2 28101.009} C_VEL
LIN {X 0,Y 592.529,Z 546.026,A -85,B 0,C 180,E1 28097.936,E2 28097.936} C_VEL
LIN {X 0,Y 592.326,Z 582.99,A -85,B 0,C 180,E1 28094.817,E2 28094.817} C_VEL
LIN {X 0,Y 592.301,Z 602.631,A -85,B 0,C 180,E1 28093.204,E2 28093.204} C_VEL
LIN {X 0,Y 592.379,Z 744.346,A -85,B 0,C 180,E1 28091.43,E2 28091.43} C_VEL
LIN {X 0,Y 592.336,Z 761.107,A -85,B 0,C 180,E1 28091.028,E2 28091.028} C_VEL
LIN {X 0,Y 592.276,Z 775.66,A -85,B 0,C 180,E1 28090.505,E2 28090.505} C_VEL
LIN {X 0,Y 592.219,Z 790.043,A -85,B 0,C 180,E1 28089.818,E2 28089.818} C_VEL
LIN {X 0,Y 592.151,Z 804.293,A -85,B 0,C 180,E1 28088.937,E2 28088.937} C_VEL
LIN {X 0,Y 592.078,Z 817.413,A -85,B 0,C 180,E1 28087.911,E2 28087.911} C_VEL
LIN {X 0,Y 592.021,Z 829.846,A -85,B 0,C 180,E1 28086.692,E2 28086.692} C_VEL
LIN {X 0,Y 591.975,Z 840.108,A -85,B 0,C 180,E1 28085.428,E2 28085.428} C_VEL
LIN {X 0,Y 591.945,Z 849.489,A -85,B 0,C 180,E1 28083.971,E2 28083.971} C_VEL
LIN {X 0,Y 591.926,Z 856.593,A -85,B 0,C 180,E1 28082.517,E2 28082.517} C_VEL
LIN {X 0,Y 591.918,Z 862.169,A -85,B 0,C 180,E1 28080.968,E2 28080.968} C_VEL
LIN {X 0,Y 591.915,Z 865.799,A -85,B 0,C 180,E1 28079.419,E2 28079.419} C_VEL
LIN {X 0,Y 591.914,Z 867.667,A -85,B 0,C 180,E1 28077.87,E2 28077.87} C_VEL
LIN {X 0,Y 591.915,Z 867.855,A -85,B 0,C 180,E1 28076.32,E2 28076.32} C_VEL
LIN {X 0,Y 591.916,Z 866.247,A -85,B 0,C 180,E1 28074.767,E2 28074.767} C_VEL
LIN {X 0,Y 591.917,Z 862.922,A -85,B 0,C 180,E1 28073.209,E2 28073.209} C_VEL
LIN {X 0,Y 591.924,Z 857.653,A -85,B 0,C 180,E1 28071.647,E2 28071.647} C_VEL
LIN {X 0,Y 591.938,Z 850.758,A -85,B 0,C 180,E1 28070.177,E2 28070.177} C_VEL
LIN {X 0,Y 591.969,Z 842.393,A -85,B 0,C 180,E1 28068.8,E2 28068.8} C_VEL
LIN {X 0,Y 592.006,Z 832.105,A -85,B 0,C 180,E1 28067.478,E2 28067.478} C_VEL
LIN {X 0,Y 592.069,Z 820.502,A -85,B 0,C 180,E1 28066.275,E2 28066.275} C_VEL
LIN {X 0,Y 592.132,Z 807.137,A -85,B 0,C 180,E1 28065.178,E2 28065.178} C_VEL
LIN {X 0,Y 592.207,Z 793.369,A -85,B 0,C 180,E1 28064.277,E2 28064.277} C_VEL
LIN {X 0,Y 592.268,Z 777.438,A -85,B 0,C 180,E1 28063.479,E2 28063.479} C_VEL
LIN {X 0,Y 592.322,Z 762.291,A -85,B 0,C 180,E1 28062.92,E2 28062.92} C_VEL
LIN {X 0,Y 592.37,Z 745.255,A -85,B 0,C 180,E1 28062.497,E2 28062.497} C_VEL
LIN {X 0,Y 592.437,Z 706.566,A -85,B 0,C 180,E1 28061.991,E2 28061.991} C_VEL
LIN {X 0,Y 592.252,Z 602.284,A -85,B 0,C 180,E1 28060.7,E2 28060.7} C_VEL
LIN {X 0,Y 592.416,Z 563.715,A -85,B 0,C 180,E1 28057.473,E2 28057.473} C_VEL
LIN {X 0,Y 592.557,Z 529.018,A -85,B 0,C 180,E1 28054.515,E2 28054.515} C_VEL
LIN {X 0,Y 592.763,Z 507.662,A -85,B 0,C 180,E1 28052.636,E2 28052.636} C_VEL
LIN {X 0,Y 594.734,Z 474.155,A -85,B 0,C 180,E1 28049.264,E2 28049.264} C_VEL
LIN {X 0,Y 595.189,Z 452.162,A -85,B 0,C 180,E1 28046.783,E2 28046.783} C_VEL
LIN {X 0,Y 595.199,Z 449.287,A -85,B 0,C 180,E1 28046.432,E2 28046.432} C_VEL
LIN {X 0,Y 593.311,Z 445.191,A -85,B 0,C 180,E1 28045.666,E2 28045.666} C_VEL
LIN {X 0,Y 592.03,Z 441.742,A -85,B 0,C 180,E1 28044.996,E2 28044.996} C_VEL
LIN {X 0,Y 592.033,Z 441.737,A -85,B 0,C 180,E1 28041.698,E2 28041.698} C_VEL
LIN {X 0,Y 592.001,Z 441.744,A -85,B 0,C 180,E1 28038.542,E2 28038.542} C_VEL
LIN {X 0,Y 591.997,Z 441.795,A -85,B 0,C 180,E1 28036.075,E2 28036.075} C_VEL
LIN {X 0,Y 593.084,Z 444.854,A -85,B 0,C 180,E1 28035.738,E2 28035.738} C_VEL
LIN {X 0,Y 594.263,Z 447.47,A -85,B 0,C 180,E1 28035.444,E2 28035.444} C_VEL
LIN {X 0,Y 593.55,Z 477.074,A -85,B 0,C 180,E1 28033.55,E2 28033.55} C_VEL
LIN {X 0,Y 593.582,Z 534.066,A -85,B 0,C 180,E1 28030.217,E2 28030.217} C_VEL
LIN {X 0,Y 595.379,Z 549.37,A -85,B 0,C 180,E1 28029.269,E2 28029.269} C_VEL
LIN {X 0,Y 597.408,Z 557.491,A -85,B 0,C 180,E1 28028.63,E2 28028.63} C_VEL
LIN {X 0,Y 599.328,Z 562.429,A -85,B 0,C 180,E1 28028.054,E2 28028.054} C_VEL
LIN {X 0,Y 601.097,Z 565.157,A -85,B 0,C 180,E1 28027.492,E2 28027.492} C_VEL
LIN {X 0,Y 602.481,Z 566.078,A -85,B 0,C 180,E1 28026.925,E2 28026.925} C_VEL
LIN {X 0,Y 603.218,Z 565.251,A -85,B 0,C 180,E1 28026.399,E2 28026.399} C_VEL
LIN {X 0,Y 603.2,Z 562.867,A -85,B 0,C 180,E1 28025.914,E2 28025.914} C_VEL
LIN {X 0,Y 602.39,Z 558.935,A -85,B 0,C 180,E1 28025.502,E2 28025.502} C_VEL
LIN {X 0,Y 600.927,Z 553.581,A -85,B 0,C 180,E1 28025.207,E2 28025.207} C_VEL
LIN {X 0,Y 599.383,Z 545.839,A -85,B 0,C 180,E1 28024.998,E2 28024.998} C_VEL
LIN {X 0,Y 598.653,Z 535.258,A -85,B 0,C 180,E1 28024.898,E2 28024.898} C_VEL
LIN {X 0,Y 598.487,Z 450.597,A -85,B 0,C 180,E1 28024.875,E2 28024.875} C_VEL
LIN {X 0,Y 597.204,Z 448.628,A -85,B 0,C 180,E1 28024.698,E2 28024.698} C_VEL
LIN {X 0,Y 595.218,Z 450.373,A -85,B 0,C 180,E1 28024.421,E2 28024.421} C_VEL
LIN {X 0,Y 593.931,Z 450.331,A -85,B 0,C 180,E1 28024.229,E2 28024.229} C_VEL
LIN {X 0,Y 593.621,Z 498.992,A -85,B 0,C 180,E1 28021.169,E2 28021.169} C_VEL
LIN {X 0,Y 593.341,Z 544.227,A -85,B 0,C 180,E1 28018.427,E2 28018.427} C_VEL
LIN {X 0,Y 593.692,Z 549.826,A -85,B 0,C 180,E1 28018.333,E2 28018.333} C_VEL
LIN {X 0,Y 593.334,Z 806.458,A -85,B 0,C 180,E1 28014.92,E2 28014.92} C_VEL
LIN {X 0,Y 593.228,Z 827.385,A -85,B 0,C 180,E1 28014.452,E2 28014.452} C_VEL
LIN {X 0,Y 593.103,Z 847.531,A -85,B 0,C 180,E1 28013.813,E2 28013.813} C_VEL
LIN {X 0,Y 592.95,Z 866.611,A -85,B 0,C 180,E1 28013.03,E2 28013.03} C_VEL
LIN {X 0,Y 592.808,Z 885.067,A -85,B 0,C 180,E1 28012.094,E2 28012.094} C_VEL
LIN {X 0,Y 592.645,Z 904.016,A -85,B 0,C 180,E1 28010.924,E2 28010.924} C_VEL
LIN {X 0,Y 592.49,Z 921.553,A -85,B 0,C 180,E1 28009.623,E2 28009.623} C_VEL
LIN {X 0,Y 592.337,Z 938.494,A -85,B 0,C 180,E1 28008.133,E2 28008.133} C_VEL
LIN {X 0,Y 592.212,Z 953.433,A -85,B 0,C 180,E1 28006.579,E2 28006.579} C_VEL
LIN {X 0,Y 592.109,Z 967.37,A -85,B 0,C 180,E1 28004.873,E2 28004.873} C_VEL
LIN {X 0,Y 592.029,Z 979.012,A -85,B 0,C 180,E1 28003.18,E2 28003.18} C_VEL
LIN {X 0,Y 591.979,Z 989.326,A -85,B 0,C 180,E1 28001.398,E2 28001.398} C_VEL
LIN {X 0,Y 591.943,Z 998.254,A -85,B 0,C 180,E1 27999.529,E2 27999.529} C_VEL
LIN {X 0,Y 591.925,Z 1005.683,A -85,B 0,C 180,E1 27997.572,E2 27997.572} C_VEL
LIN {X 0,Y 591.913,Z 1011.25,A -85,B 0,C 180,E1 27995.623,E2 27995.623} C_VEL
LIN {X 0,Y 591.909,Z 1015.088,A -85,B 0,C 180,E1 27993.681,E2 27993.681} C_VEL
LIN {X 0,Y 591.903,Z 1017.377,A -85,B 0,C 180,E1 27991.646,E2 27991.646} C_VEL
LIN {X 0,Y 591.9,Z 1017.918,A -85,B 0,C 180,E1 27989.613,E2 27989.613} C_VEL
LIN {X 0,Y 591.907,Z 1016.846,A -85,B 0,C 180,E1 27987.677,E2 27987.677} C_VEL
LIN {X 0,Y 591.913,Z 1013.972,A -85,B 0,C 180,E1 27985.641,E2 27985.641} C_VEL
LIN {X 0,Y 591.922,Z 1009.48,A -85,B 0,C 180,E1 27983.697,E2 27983.697} C_VEL
LIN {X 0,Y 591.934,Z 1003.274,A -85,B 0,C 180,E1 27981.746,E2 27981.746} C_VEL
LIN {X 0,Y 591.953,Z 995.186,A -85,B 0,C 180,E1 27979.785,E2 27979.785} C_VEL
LIN {X 0,Y 591.999,Z 985.563,A -85,B 0,C 180,E1 27977.912,E2 27977.912} C_VEL
LIN {X 0,Y 592.064,Z 974.51,A -85,B 0,C 180,E1 27976.126,E2 27976.126} C_VEL
LIN {X 0,Y 592.152,Z 961.126,A -85,B 0,C 180,E1 27974.327,E2 27974.327} C_VEL
LIN {X 0,Y 592.272,Z 946.48,A -85,B 0,C 180,E1 27972.664,E2 27972.664} C_VEL
LIN {X 0,Y 592.406,Z 930.609,A -85,B 0,C 180,E1 27971.143,E2 27971.143} C_VEL
LIN {X 0,Y 592.559,Z 913.419,A -85,B 0,C 180,E1 27969.746,E2 27969.746} C_VEL
LIN {X 0,Y 592.71,Z 895.556,A -85,B 0,C 180,E1 27968.528,E2 27968.528} C_VEL
LIN {X 0,Y 592.856,Z 877.308,A -85,B 0,C 180,E1 27967.491,E2 27967.491} C_VEL
LIN {X 0,Y 593.025,Z 858.303,A -85,B 0,C 180,E1 27966.606,E2 27966.606} C_VEL
LIN {X 0,Y 593.168,Z 838.607,A -85,B 0,C 180,E1 27965.88,E2 27965.88} C_VEL
LIN {X 0,Y 593.271,Z 818.47,A -85,B 0,C 180,E1 27965.324,E2 27965.324} C_VEL
LIN {X 0,Y 593.352,Z 797.383,A -85,B 0,C 180,E1 27964.939,E2 27964.939} C_VEL
LIN {X 0,Y 593.693,Z 549.404,A -85,B 0,C 180,E1 27961.661,E2 27961.661} C_VEL
LIN {X 0,Y 593.295,Z 543.932,A -85,B 0,C 180,E1 27961.567,E2 27961.567} C_VEL
LIN {X 0,Y 593.639,Z 495.889,A -85,B 0,C 180,E1 27958.639,E2 27958.639} C_VEL
LIN {X 0,Y 593.944,Z 450.173,A -85,B 0,C 180,E1 27955.759,E2 27955.759} C_VEL
LIN {X 0,Y 595.496,Z 450.242,A -85,B 0,C 180,E1 27955.54,E2 27955.54} C_VEL
LIN {X 0,Y 597.34,Z 448.665,A -85,B 0,C 180,E1 27955.283,E2 27955.283} C_VEL
LIN {X 0,Y 598.615,Z 450.776,A -85,B 0,C 180,E1 27955.108,E2 27955.108} C_VEL
LIN {X 0,Y 598.767,Z 538.666,A -85,B 0,C 180,E1 27955.087,E2 27955.087} C_VEL
LIN {X 0,Y 599.734,Z 548.214,A -85,B 0,C 180,E1 27954.955,E2 27954.955} C_VEL
LIN {X 0,Y 601.483,Z 555.555,A -85,B 0,C 180,E1 27954.707,E2 27954.707} C_VEL
LIN {X 0,Y 602.74,Z 560.368,A -85,B 0,C 180,E1 27954.374,E2 27954.374} C_VEL
LIN {X 0,Y 603.287,Z 563.656,A -85,B 0,C 180,E1 27953.96,E2 27953.96} C_VEL
LIN {X 0,Y 603.096,Z 565.621,A -85,B 0,C 180,E1 27953.475,E2 27953.475} C_VEL
LIN {X 0,Y 602.193,Z 566.017,A -85,B 0,C 180,E1 27952.936,E2 27952.936} C_VEL
LIN {X 0,Y 600.606,Z 564.54,A -85,B 0,C 180,E1 27952.341,E2 27952.341} C_VEL
LIN {X 0,Y 598.774,Z 561.25,A -85,B 0,C 180,E1 27951.782,E2 27951.782} C_VEL
LIN {X 0,Y 596.783,Z 555.294,A -85,B 0,C 180,E1 27951.175,E2 27951.175} C_VEL
LIN {X 0,Y 594.954,Z 545.355,A -85,B 0,C 180,E1 27950.41,E2 27950.41} C_VEL
LIN {X 0,Y 594.223,Z 527.45,A -85,B 0,C 180,E1 27949.186,E2 27949.186} C_VEL
LIN {X 0,Y 594.578,Z 490.138,A -85,B 0,C 180,E1 27946.678,E2 27946.678} C_VEL
LIN {X 0,Y 594.988,Z 448.985,A -85,B 0,C 180,E1 27943.783,E2 27943.783} C_VEL
LIN {X 0,Y 593.142,Z 444.978,A -85,B 0,C 180,E1 27943.32,E2 27943.32} C_VEL
LIN {X 0,Y 592.031,Z 441.744,A -85,B 0,C 180,E1 27942.946,E2 27942.946} C_VEL
LIN {X 0,Y 592.032,Z 441.744,A -85,B 0,C 180,E1 27939.636,E2 27939.636} C_VEL
LIN {X 0,Y 592.015,Z 441.742,A -85,B 0,C 180,E1 27936.476,E2 27936.476} C_VEL
LIN {X 0,Y 592.017,Z 441.741,A -85,B 0,C 180,E1 27933.28,E2 27933.28} C_VEL
LIN {X 0,Y 592.041,Z 441.738,A -85,B 0,C 180,E1 27929.961,E2 27929.961} C_VEL
LIN {X 0,Y 592.001,Z 441.743,A -85,B 0,C 180,E1 27926.691,E2 27926.691} C_VEL
LIN {X 0,Y 592.029,Z 441.738,A -85,B 0,C 180,E1 27923.489,E2 27923.489} C_VEL
LIN {X 0,Y 591.981,Z 441.743,A -85,B 0,C 180,E1 27920.382,E2 27920.382} C_VEL
LIN {X 0,Y 592.01,Z 441.74,A -85,B 0,C 180,E1 27917.075,E2 27917.075} C_VEL
LIN {X 0,Y 592.007,Z 441.74,A -85,B 0,C 180,E1 27913.976,E2 27913.976} C_VEL
LIN {X 0,Y 591.98,Z 441.743,A -85,B 0,C 180,E1 27910.582,E2 27910.582} C_VEL
LIN {X 0,Y 592.03,Z 441.737,A -85,B 0,C 180,E1 27907.472,E2 27907.472} C_VEL
LIN {X 0,Y 591.989,Z 441.743,A -85,B 0,C 180,E1 27904.262,E2 27904.262} C_VEL
LIN {X 0,Y 592.032,Z 441.737,A -85,B 0,C 180,E1 27900.968,E2 27900.968} C_VEL
LIN {X 0,Y 592.014,Z 441.741,A -85,B 0,C 180,E1 27897.774,E2 27897.774} C_VEL
LIN {X 0,Y 592.011,Z 441.743,A -85,B 0,C 180,E1 27894.573,E2 27894.573} C_VEL
LIN {X 0,Y 592.036,Z 441.742,A -85,B 0,C 180,E1 27891.453,E2 27891.453} C_VEL
LIN {X 0,Y 592.029,Z 441.74,A -85,B 0,C 180,E1 27890.073,E2 27890.073} C_VEL
LIN {X 0,Y 591.038,Z 441.868,A -85,B 0,C 180,E1 27889.327,E2 27889.327} C_VEL
LIN {X 0,Y 584.581,Z 442.663,A -85,B 0,C 180,E1 27887.236,E2 27887.236} C_VEL
LIN {X 0,Y 584.082,Z 442.729,A -85,B 0,C 180,E1 27886.691,E2 27886.691} C_VEL
LIN {X 0,Y 584.079,Z 442.731,A -85,B 0,C 180,E1 27883.462,E2 27883.462} C_VEL
LIN {X 0,Y 584.099,Z 442.727,A -85,B 0,C 180,E1 27880.188,E2 27880.188} C_VEL
LIN {X 0,Y 584.06,Z 442.73,A -85,B 0,C 180,E1 27876.919,E2 27876.919} C_VEL
LIN {X 0,Y 584.086,Z 442.728,A -85,B 0,C 180,E1 27873.681,E2 27873.681} C_VEL
LIN {X 0,Y 584.05,Z 442.731,A -85,B 0,C 180,E1 27870.572,E2 27870.572} C_VEL
LIN {X 0,Y 584.064,Z 442.73,A -85,B 0,C 180,E1 27867.251,E2 27867.251} C_VEL
LIN {X 0,Y 584.077,Z 442.728,A -85,B 0,C 180,E1 27864.165,E2 27864.165} C_VEL
LIN {X 0,Y 584.041,Z 442.732,A -85,B 0,C 180,E1 27860.823,E2 27860.823} C_VEL
LIN {X 0,Y 584.095,Z 442.726,A -85,B 0,C 180,E1 27857.688,E2 27857.688} C_VEL
LIN {X 0,Y 584.053,Z 442.731,A -85,B 0,C 180,E1 27854.441,E2 27854.441} C_VEL
LIN {X 0,Y 584.086,Z 442.729,A -85,B 0,C 180,E1 27851.227,E2 27851.227} C_VEL
LIN {X 0,Y 584.081,Z 442.731,A -85,B 0,C 180,E1 27848.043,E2 27848.043} C_VEL
LIN {X 0,Y 584.08,Z 442.733,A -85,B 0,C 180,E1 27844.872,E2 27844.872} C_VEL
LIN {X 0,Y 584.079,Z 442.748,A -85,B 0,C 180,E1 27842.84,E2 27842.84} C_VEL
LIN {X 0,Y 586.338,Z 449.936,A -85,B 0,C 180,E1 27842.143,E2 27842.143} C_VEL
LIN {X 0,Y 585.887,Z 491.187,A -85,B 0,C 180,E1 27839.046,E2 27839.046} C_VEL
LIN {X 0,Y 585.952,Z 495.481,A -85,B 0,C 180,E1 27838.756,E2 27838.756} C_VEL
LIN {X 0,Y 586.705,Z 500.76,A -85,B 0,C 180,E1 27838.644,E2 27838.644} C_VEL
LIN {X 0,Y 586.125,Z 740.823,A -85,B 0,C 180,E1 27835.437,E2 27835.437} C_VEL
LIN {X 0,Y 586.024,Z 763.605,A -85,B 0,C 180,E1 27835.062,E2 27835.062} C_VEL
LIN {X 0,Y 585.839,Z 784.474,A -85,B 0,C 180,E1 27834.526,E2 27834.526} C_VEL
LIN {X 0,Y 585.66,Z 803.399,A -85,B 0,C 180,E1 27833.866,E2 27833.866} C_VEL
LIN {X 0,Y 585.436,Z 822.981,A -85,B 0,C 180,E1 27832.993,E2 27832.993} C_VEL
LIN {X 0,Y 585.199,Z 841.427,A -85,B 0,C 180,E1 27831.973,E2 27831.973} C_VEL
LIN {X 0,Y 584.944,Z 859.501,A -85,B 0,C 180,E1 27830.771,E2 27830.771} C_VEL
LIN {X 0,Y 584.7,Z 876.621,A -85,B 0,C 180,E1 27829.417,E2 27829.417} C_VEL
LIN {X 0,Y 584.487,Z 893.027,A -85,B 0,C 180,E1 27827.882,E2 27827.882} C_VEL
LIN {X 0,Y 584.307,Z 907.663,A -85,B 0,C 180,E1 27826.264,E2 27826.264} C_VEL
LIN {X 0,Y 584.164,Z 921.378,A -85,B 0,C 180,E1 27824.471,E2 27824.471} C_VEL
LIN {X 0,Y 584.062,Z 933.142,A -85,B 0,C 180,E1 27822.634,E2 27822.634} C_VEL
LIN {X 0,Y 583.99,Z 942.669,A -85,B 0,C 180,E1 27820.855,E2 27820.855} C_VEL
LIN {X 0,Y 583.944,Z 951.186,A -85,B 0,C 180,E1 27818.896,E2 27818.896} C_VEL
LIN {X 0,Y 583.916,Z 957.674,A -85,B 0,C 180,E1 27816.983,E2 27816.983} C_VEL
LIN {X 0,Y 583.907,Z 962.665,A -85,B 0,C 180,E1 27815.01,E2 27815.01} C_VEL
LIN {X 0,Y 583.905,Z 966.005,A -85,B 0,C 180,E1 27813.042,E2 27813.042} C_VEL
LIN {X 0,Y 583.907,Z 967.74,A -85,B 0,C 180,E1 27811.079,E2 27811.079} C_VEL
LIN {X 0,Y 583.912,Z 967.795,A -85,B 0,C 180,E1 27809.018,E2 27809.018} C_VEL
LIN {X 0,Y 583.912,Z 966.219,A -85,B 0,C 180,E1 27807.055,E2 27807.055} C_VEL
LIN {X 0,Y 583.91,Z 962.85,A -85,B 0,C 180,E1 27804.989,E2 27804.989} C_VEL
LIN {X 0,Y 583.921,Z 957.945,A -85,B 0,C 180,E1 27803.016,E2 27803.016} C_VEL
LIN {X 0,Y 583.943,Z 951.269,A -85,B 0,C 180,E1 27801.035,E2 27801.035} C_VEL
LIN {X 0,Y 583.983,Z 943.079,A -85,B 0,C 180,E1 27799.144,E2 27799.144} C_VEL
LIN {X 0,Y 584.059,Z 933.519,A -85,B 0,C 180,E1 27797.342,E2 27797.342} C_VEL
LIN {X 0,Y 584.158,Z 921.998,A -85,B 0,C 180,E1 27795.528,E2 27795.528} C_VEL
LIN {X 0,Y 584.3,Z 908.976,A -85,B 0,C 180,E1 27793.803,E2 27793.803} C_VEL
LIN {X 0,Y 584.475,Z 894.407,A -85,B 0,C 180,E1 27792.168,E2 27792.168} C_VEL
LIN {X 0,Y 584.687,Z 878.75,A -85,B 0,C 180,E1 27790.676,E2 27790.676} C_VEL
LIN {X 0,Y 584.921,Z 862.146,A -85,B 0,C 180,E1 27789.329,E2 27789.329} C_VEL
LIN {X 0,Y 585.174,Z 844.056,A -85,B 0,C 180,E1 27788.094,E2 27788.094} C_VEL
LIN {X 0,Y 585.399,Z 824.918,A -85,B 0,C 180,E1 27787.016,E2 27787.016} C_VEL
LIN {X 0,Y 585.618,Z 805.516,A -85,B 0,C 180,E1 27786.131,E2 27786.131} C_VEL
LIN {X 0,Y 585.837,Z 785.082,A -85,B 0,C 180,E1 27785.403,E2 27785.403} C_VEL
LIN {X 0,Y 586.021,Z 764.307,A -85,B 0,C 180,E1 27784.862,E2 27784.862} C_VEL
LIN {X 0,Y 586.125,Z 741.78,A -85,B 0,C 180,E1 27784.485,E2 27784.485} C_VEL
LIN {X 0,Y 586.634,Z 502.798,A -85,B 0,C 180,E1 27781.29,E2 27781.29} C_VEL
LIN {X 0,Y 585.273,Z 497.392,A -85,B 0,C 180,E1 27781.129,E2 27781.129} C_VEL
LIN {X 0,Y 585.604,Z 468.338,A -85,B 0,C 180,E1 27777.873,E2 27777.873} C_VEL
LIN {X 0,Y 585.754,Z 448.648,A -85,B 0,C 180,E1 27775.597,E2 27775.597} C_VEL
LIN {X 0,Y 584.088,Z 442.728,A -85,B 0,C 180,E1 27774.74,E2 27774.74} C_VEL
LIN {X 0,Y 584.068,Z 442.733,A -85,B 0,C 180,E1 27771.58,E2 27771.58} C_VEL
LIN {X 0,Y 584.069,Z 442.726,A -85,B 0,C 180,E1 27768.246,E2 27768.246} C_VEL
LIN {X 0,Y 584.094,Z 442.728,A -85,B 0,C 180,E1 27765.01,E2 27765.01} C_VEL
LIN {X 0,Y 584.072,Z 442.727,A -85,B 0,C 180,E1 27761.753,E2 27761.753} C_VEL
LIN {X 0,Y 584.088,Z 442.725,A -85,B 0,C 180,E1 27758.527,E2 27758.527} C_VEL
LIN {X 0,Y 584.094,Z 442.733,A -85,B 0,C 180,E1 27755.232,E2 27755.232} C_VEL
LIN {X 0,Y 584.093,Z 442.726,A -85,B 0,C 180,E1 27751.889,E2 27751.889} C_VEL
LIN {X 0,Y 584.071,Z 442.732,A -85,B 0,C 180,E1 27748.753,E2 27748.753} C_VEL
LIN {X 0,Y 584.118,Z 442.911,A -85,B 0,C 180,E1 27747.693,E2 27747.693} C_VEL
LIN {X 0,Y 585.968,Z 449.718,A -85,B 0,C 180,E1 27746.939,E2 27746.939} C_VEL
LIN {X 0,Y 585.681,Z 480.634,A -85,B 0,C 180,E1 27744.08,E2 27744.08} C_VEL
LIN {X 0,Y 585.117,Z 514.225,A -85,B 0,C 180,E1 27741.03,E2 27741.03} C_VEL
LIN {X 0,Y 584.821,Z 548.928,A -85,B 0,C 180,E1 27737.975,E2 27737.975} C_VEL
LIN {X 0,Y 584.552,Z 585.895,A -85,B 0,C 180,E1 27734.816,E2 27734.816} C_VEL
LIN {X 0,Y 584.511,Z 602.715,A -85,B 0,C 180,E1 27733.426,E2 27733.426} C_VEL
LIN {X 0,Y 584.807,Z 612.603,A -85,B 0,C 180,E1 27733.293,E2 27733.293} C_VEL
LIN {X 0,Y 584.626,Z 744.017,A -85,B 0,C 180,E1 27731.63,E2 27731.63} C_VEL
LIN {X 0,Y 584.559,Z 761.186,A -85,B 0,C 180,E1 27731.216,E2 27731.216} C_VEL
LIN {X 0,Y 584.469,Z 775.887,A -85,B 0,C 180,E1 27730.679,E2 27730.679} C_VEL
LIN {X 0,Y 584.373,Z 790.807,A -85,B 0,C 180,E1 27729.951,E2 27729.951} C_VEL
LIN {X 0,Y 584.266,Z 804.855,A -85,B 0,C 180,E1 27729.059,E2 27729.059} C_VEL
LIN {X 0,Y 584.166,Z 817.319,A -85,B 0,C 180,E1 27728.068,E2 27728.068} C_VEL
LIN {X 0,Y 584.078,Z 829.737,A -85,B 0,C 180,E1 27726.838,E2 27726.838} C_VEL
LIN {X 0,Y 584.008,Z 839.691,A -85,B 0,C 180,E1 27725.6,E2 27725.6} C_VEL
LIN {X 0,Y 583.963,Z 848.602,A -85,B 0,C 180,E1 27724.222,E2 27724.222} C_VEL
LIN {X 0,Y 583.933,Z 855.937,A -85,B 0,C 180,E1 27722.748,E2 27722.748} C_VEL
LIN {X 0,Y 583.922,Z 861.397,A -85,B 0,C 180,E1 27721.276,E2 27721.276} C_VEL
LIN {X 0,Y 583.916,Z 865.543,A -85,B 0,C 180,E1 27719.608,E2 27719.608} C_VEL
LIN {X 0,Y 583.915,Z 867.557,A -85,B 0,C 180,E1 27718.038,E2 27718.038} C_VEL
LIN {X 0,Y 583.916,Z 867.878,A -85,B 0,C 180,E1 27716.368,E2 27716.368} C_VEL
LIN {X 0,Y 583.916,Z 866.33,A -85,B 0,C 180,E1 27714.793,E2 27714.793} C_VEL
LIN {X 0,Y 583.919,Z 863.066,A -85,B 0,C 180,E1 27713.215,E2 27713.215} C_VEL
LIN {X 0,Y 583.929,Z 857.882,A -85,B 0,C 180,E1 27711.631,E2 27711.631} C_VEL
LIN {X 0,Y 583.949,Z 851.568,A -85,B 0,C 180,E1 27710.241,E2 27710.241} C_VEL
LIN {X 0,Y 583.989,Z 843.323,A -85,B 0,C 180,E1 27708.829,E2 27708.829} C_VEL
LIN {X 0,Y 584.048,Z 833.762,A -85,B 0,C 180,E1 27707.543,E2 27707.543} C_VEL
LIN {X 0,Y 584.122,Z 822.633,A -85,B 0,C 180,E1 27706.337,E2 27706.337} C_VEL
LIN {X 0,Y 584.229,Z 809.918,A -85,B 0,C 180,E1 27705.227,E2 27705.227} C_VEL
LIN {X 0,Y 584.315,Z 796.759,A -85,B 0,C 180,E1 27704.314,E2 27704.314} C_VEL
LIN {X 0,Y 584.418,Z 783,A -85,B 0,C 180,E1 27703.552,E2 27703.552} C_VEL
LIN {X 0,Y 584.527,Z 767.083,A -85,B 0,C 180,E1 27702.89,E2 27702.89} C_VEL
LIN {X 0,Y 584.585,Z 751.732,A -85,B 0,C 180,E1 27702.442,E2 27702.442} C_VEL
LIN {X 0,Y 584.653,Z 735.079,A -85,B 0,C 180,E1 27702.142,E2 27702.142} C_VEL
LIN {X 0,Y 584.583,Z 603.29,A -85,B 0,C 180,E1 27700.494,E2 27700.494} C_VEL
LIN {X 0,Y 584.452,Z 602.088,A -85,B 0,C 180,E1 27700.461,E2 27700.461} C_VEL
LIN {X 0,Y 584.684,Z 563.175,A -85,B 0,C 180,E1 27697.158,E2 27697.158} C_VEL
LIN {X 0,Y 584.956,Z 531.771,A -85,B 0,C 180,E1 27694.423,E2 27694.423} C_VEL
LIN {X 0,Y 586.783,Z 497.377,A -85,B 0,C 180,E1 27691.002,E2 27691.002} C_VEL
LIN {X 0,Y 588.283,Z 474.901,A -85,B 0,C 180,E1 27688.662,E2 27688.662} C_VEL
LIN {X 0,Y 589.042,Z 454.148,A -85,B 0,C 180,E1 27686.243,E2 27686.243} C_VEL
LIN {X 0,Y 587.628,Z 450.786,A -85,B 0,C 180,E1 27685.605,E2 27685.605} C_VEL
LIN {X 0,Y 585.812,Z 446.773,A -85,B 0,C 180,E1 27684.768,E2 27684.768} C_VEL
LIN {X 0,Y 584.275,Z 443.725,A -85,B 0,C 180,E1 27684.042,E2 27684.042} C_VEL
LIN {X 0,Y 584.096,Z 442.729,A -85,B 0,C 180,E1 27683.803,E2 27683.803} C_VEL
LIN {X 0,Y 584.07,Z 442.733,A -85,B 0,C 180,E1 27680.54,E2 27680.54} C_VEL
LIN {X 0,Y 584.099,Z 442.731,A -85,B 0,C 180,E1 27677.323,E2 27677.323} C_VEL
LIN {X 0,Y 584.106,Z 442.945,A -85,B 0,C 180,E1 27676.861,E2 27676.861} C_VEL
LIN {X 0,Y 585.464,Z 446.375,A -85,B 0,C 180,E1 27676.374,E2 27676.374} C_VEL
LIN {X 0,Y 586.513,Z 448.627,A -85,B 0,C 180,E1 27676.066,E2 27676.066} C_VEL
LIN {X 0,Y 587.728,Z 451.157,A -85,B 0,C 180,E1 27675.744,E2 27675.744} C_VEL
LIN {X 0,Y 586.585,Z 478.201,A -85,B 0,C 180,E1 27673.928,E2 27673.928} C_VEL
LIN {X 0,Y 585.826,Z 519.972,A -85,B 0,C 180,E1 27671.405,E2 27671.405} C_VEL
LIN {X 0,Y 586.642,Z 541.566,A -85,B 0,C 180,E1 27670.11,E2 27670.11} C_VEL
LIN {X 0,Y 588.509,Z 554.142,A -85,B 0,C 180,E1 27669.304,E2 27669.304} C_VEL
LIN {X 0,Y 591.43,Z 563.382,A -85,B 0,C 180,E1 27668.644,E2 27668.644} C_VEL
LIN {X 0,Y 593.991,Z 568.337,A -85,B 0,C 180,E1 27668.154,E2 27668.154} C_VEL
LIN {X 0,Y 596.757,Z 571.815,A -85,B 0,C 180,E1 27667.58,E2 27667.58} C_VEL
LIN {X 0,Y 598.826,Z 573.272,A -85,B 0,C 180,E1 27667.05,E2 27667.05} C_VEL
LIN {X 0,Y 600.416,Z 573.189,A -85,B 0,C 180,E1 27666.455,E2 27666.455} C_VEL
LIN {X 0,Y 601.029,Z 571.398,A -85,B 0,C 180,E1 27665.877,E2 27665.877} C_VEL
LIN {X 0,Y 600.535,Z 568.073,A -85,B 0,C 180,E1 27665.365,E2 27665.365} C_VEL
LIN {X 0,Y 599.028,Z 563.488,A -85,B 0,C 180,E1 27664.961,E2 27664.961} C_VEL
LIN {X 0,Y 596.6,Z 556.333,A -85,B 0,C 180,E1 27664.614,E2 27664.614} C_VEL
LIN {X 0,Y 594.937,Z 547.561,A -85,B 0,C 180,E1 27664.381,E2 27664.381} C_VEL
LIN {X 0,Y 594.134,Z 536.406,A -85,B 0,C 180,E1 27664.268,E2 27664.268} C_VEL
LIN {X 0,Y 594.02,Z 464.466,A -85,B 0,C 180,E1 27664.252,E2 27664.252} C_VEL
LIN {X 0,Y 590.525,Z 471.122,A -85,B 0,C 180,E1 27663.751,E2 27663.751} C_VEL
LIN {X 0,Y 588.245,Z 473.612,A -85,B 0,C 180,E1 27663.417,E2 27663.417} C_VEL
LIN {X 0,Y 586.771,Z 473.667,A -85,B 0,C 180,E1 27663.19,E2 27663.19} C_VEL
LIN {X 0,Y 586.275,Z 523.963,A -85,B 0,C 180,E1 27660.037,E2 27660.037} C_VEL
LIN {X 0,Y 586.137,Z 544.503,A -85,B 0,C 180,E1 27658.805,E2 27658.805} C_VEL
LIN {X 0,Y 586.648,Z 549.826,A -85,B 0,C 180,E1 27658.704,E2 27658.704} C_VEL
LIN {X 0,Y 586.108,Z 796.31,A -85,B 0,C 180,E1 27655.409,E2 27655.409} C_VEL
LIN {X 0,Y 585.995,Z 817.529,A -85,B 0,C 180,E1 27655.024,E2 27655.024} C_VEL
LIN {X 0,Y 585.825,Z 837.713,A -85,B 0,C 180,E1 27654.47,E2 27654.47} C_VEL
LIN {X 0,Y 585.612,Z 857.013,A -85,B 0,C 180,E1 27653.763,E2 27653.763} C_VEL
LIN {X 0,Y 585.37,Z 876.301,A -85,B 0,C 180,E1 27652.867,E2 27652.867} C_VEL
LIN {X 0,Y 585.159,Z 894.741,A -85,B 0,C 180,E1 27651.817,E2 27651.817} C_VEL
LIN {X 0,Y 584.911,Z 912.952,A -85,B 0,C 180,E1 27650.567,E2 27650.567} C_VEL
LIN {X 0,Y 584.677,Z 930.015,A -85,B 0,C 180,E1 27649.169,E2 27649.169} C_VEL
LIN {X 0,Y 584.464,Z 945.98,A -85,B 0,C 180,E1 27647.626,E2 27647.626} C_VEL
LIN {X 0,Y 584.293,Z 960.289,A -85,B 0,C 180,E1 27645.993,E2 27645.993} C_VEL
LIN {X 0,Y 584.149,Z 973.098,A -85,B 0,C 180,E1 27644.27,E2 27644.27} C_VEL
LIN {X 0,Y 584.058,Z 983.826,A -85,B 0,C 180,E1 27642.558,E2 27642.558} C_VEL
LIN {X 0,Y 583.982,Z 993.34,A -85,B 0,C 180,E1 27640.756,E2 27640.756} C_VEL
LIN {X 0,Y 583.942,Z 1001.472,A -85,B 0,C 180,E1 27638.865,E2 27638.865} C_VEL
LIN {X 0,Y 583.918,Z 1007.808,A -85,B 0,C 180,E1 27636.984,E2 27636.984} C_VEL
LIN {X 0,Y 583.909,Z 1012.762,A -85,B 0,C 180,E1 27635.011,E2 27635.011} C_VEL
LIN {X 0,Y 583.907,Z 1016.065,A -85,B 0,C 180,E1 27633.043,E2 27633.043} C_VEL
LIN {X 0,Y 583.913,Z 1017.779,A -85,B 0,C 180,E1 27630.982,E2 27630.982} C_VEL
LIN {X 0,Y 583.914,Z 1017.779,A -85,B 0,C 180,E1 27629.019,E2 27629.019} C_VEL
LIN {X 0,Y 583.907,Z 1016.066,A -85,B 0,C 180,E1 27626.958,E2 27626.958} C_VEL
LIN {X 0,Y 583.909,Z 1012.763,A -85,B 0,C 180,E1 27624.991,E2 27624.991} C_VEL
LIN {X 0,Y 583.915,Z 1007.51,A -85,B 0,C 180,E1 27622.919,E2 27622.919} C_VEL
LIN {X 0,Y 583.942,Z 1001.101,A -85,B 0,C 180,E1 27621.036,E2 27621.036} C_VEL
LIN {X 0,Y 583.991,Z 992.408,A -85,B 0,C 180,E1 27619.045,E2 27619.045} C_VEL
LIN {X 0,Y 584.075,Z 982.097,A -85,B 0,C 180,E1 27617.142,E2 27617.142} C_VEL
LIN {X 0,Y 584.182,Z 970.282,A -85,B 0,C 180,E1 27615.327,E2 27615.327} C_VEL
LIN {X 0,Y 584.316,Z 956.916,A -85,B 0,C 180,E1 27613.601,E2 27613.601} C_VEL
LIN {X 0,Y 584.5,Z 941.944,A -85,B 0,C 180,E1 27611.964,E2 27611.964} C_VEL
LIN {X 0,Y 584.712,Z 925.788,A -85,B 0,C 180,E1 27610.465,E2 27610.465} C_VEL
LIN {X 0,Y 584.949,Z 908.579,A -85,B 0,C 180,E1 27609.117,E2 27609.117} C_VEL
LIN {X 0,Y 585.211,Z 890.438,A -85,B 0,C 180,E1 27607.922,E2 27607.922} C_VEL
LIN {X 0,Y 585.446,Z 872.217,A -85,B 0,C 180,E1 27606.924,E2 27606.924} C_VEL
LIN {X 0,Y 585.673,Z 852.53,A -85,B 0,C 180,E1 27606.054,E2 27606.054} C_VEL
LIN {X 0,Y 585.853,Z 832.032,A -85,B 0,C 180,E1 27605.354,E2 27605.354} C_VEL
LIN {X 0,Y 586.034,Z 811.734,A -85,B 0,C 180,E1 27604.854,E2 27604.854} C_VEL
LIN {X 0,Y 586.137,Z 785.81,A -85,B 0,C 180,E1 27604.451,E2 27604.451} C_VEL
LIN {X 0,Y 586.649,Z 547.575,A -85,B 0,C 180,E1 27601.265,E2 27601.265} C_VEL
LIN {X 0,Y 586.037,Z 543.751,A -85,B 0,C 180,E1 27601.175,E2 27601.175} C_VEL
LIN {X 0,Y 586.548,Z 495.889,A -85,B 0,C 180,E1 27598.215,E2 27598.215} C_VEL
LIN {X 0,Y 586.865,Z 473.628,A -85,B 0,C 180,E1 27596.788,E2 27596.788} C_VEL
LIN {X 0,Y 588.239,Z 473.614,A -85,B 0,C 180,E1 27596.584,E2 27596.584} C_VEL
LIN {X 0,Y 590.728,Z 470.815,A -85,B 0,C 180,E1 27596.22,E2 27596.22} C_VEL
LIN {X 0,Y 594.076,Z 464.34,A -85,B 0,C 180,E1 27595.74,E2 27595.74} C_VEL
LIN {X 0,Y 594.234,Z 539.195,A -85,B 0,C 180,E1 27595.718,E2 27595.718} C_VEL
LIN {X 0,Y 595.23,Z 549.648,A -85,B 0,C 180,E1 27595.577,E2 27595.577} C_VEL
LIN {X 0,Y 597.055,Z 557.949,A -85,B 0,C 180,E1 27595.323,E2 27595.323} C_VEL
LIN {X 0,Y 599.398,Z 564.498,A -85,B 0,C 180,E1 27594.968,E2 27594.968} C_VEL
LIN {X 0,Y 600.711,Z 568.806,A -85,B 0,C 180,E1 27594.546,E2 27594.546} C_VEL
LIN {X 0,Y 601.008,Z 571.774,A -85,B 0,C 180,E1 27594.038,E2 27594.038} C_VEL
LIN {X 0,Y 600.365,Z 573.232,A -85,B 0,C 180,E1 27593.52,E2 27593.52} C_VEL
LIN {X 0,Y 598.749,Z 573.237,A -85,B 0,C 180,E1 27592.927,E2 27592.927} C_VEL
LIN {X 0,Y 596.305,Z 571.355,A -85,B 0,C 180,E1 27592.319,E2 27592.319} C_VEL
LIN {X 0,Y 593.915,Z 568.217,A -85,B 0,C 180,E1 27591.831,E2 27591.831} C_VEL
LIN {X 0,Y 590.856,Z 561.706,A -85,B 0,C 180,E1 27591.193,E2 27591.193} C_VEL
LIN {X 0,Y 588.556,Z 551.924,A -85,B 0,C 180,E1 27590.399,E2 27590.399} C_VEL
LIN {X 0,Y 587.437,Z 536.756,A -85,B 0,C 180,E1 27589.316,E2 27589.316} C_VEL
LIN {X 0,Y 587.931,Z 494.142,A -85,B 0,C 180,E1 27586.425,E2 27586.425} C_VEL
LIN {X 0,Y 588.54,Z 452.984,A -85,B 0,C 180,E1 27583.497,E2 27583.497} C_VEL
LIN {X 0,Y 585.402,Z 446.21,A -85,B 0,C 180,E1 27582.693,E2 27582.693} C_VEL
LIN {X 0,Y 584.09,Z 442.731,A -85,B 0,C 180,E1 27582.279,E2 27582.279} C_VEL
LIN {X 0,Y 584.068,Z 442.732,A -85,B 0,C 180,E1 27579.152,E2 27579.152} C_VEL
LIN {X 0,Y 584.071,Z 442.732,A -85,B 0,C 180,E1 27575.932,E2 27575.932} C_VEL
LIN {X 0,Y 584.091,Z 442.728,A -85,B 0,C 180,E1 27572.747,E2 27572.747} C_VEL
LIN {X 0,Y 584.087,Z 442.732,A -85,B 0,C 180,E1 27569.538,E2 27569.538} C_VEL
LIN {X 0,Y 584.1,Z 442.731,A -85,B 0,C 180,E1 27566.237,E2 27566.237} C_VEL
LIN {X 0,Y 584.092,Z 442.732,A -85,B 0,C 180,E1 27562.935,E2 27562.935} C_VEL
LIN {X 0,Y 584.091,Z 442.732,A -85,B 0,C 180,E1 27559.696,E2 27559.696} C_VEL
LIN {X 0,Y 584.096,Z 442.732,A -85,B 0,C 180,E1 27556.406,E2 27556.406} C_VEL
LIN {X 0,Y 584.094,Z 442.732,A -85,B 0,C 180,E1 27553.059,E2 27553.059} C_VEL
LIN {X 0,Y 584.093,Z 442.733,A -85,B 0,C 180,E1 27549.757,E2 27549.757} C_VEL
LIN {X 0,Y 584.097,Z 442.731,A -85,B 0,C 180,E1 27546.487,E2 27546.487} C_VEL
LIN {X 0,Y 584.082,Z 442.732,A -85,B 0,C 180,E1 27543.238,E2 27543.238} C_VEL
LIN {X 0,Y 584.083,Z 442.73,A -85,B 0,C 180,E1 27540,E2 27540} C_VEL
LIN {X 0,Y 584.099,Z 442.729,A -85,B 0,C 180,E1 27536.663,E2 27536.663} C_VEL
LIN {X 0,Y 584.08,Z 442.732,A -85,B 0,C 180,E1 27533.315,E2 27533.315} C_VEL
LIN {X 0,Y 584.091,Z 442.729,A -85,B 0,C 180,E1 27530.044,E2 27530.044} C_VEL
LIN {X 0,Y 584.068,Z 442.729,A -85,B 0,C 180,E1 27526.839,E2 27526.839} C_VEL
LIN {X 0,Y 584.082,Z 442.729,A -85,B 0,C 180,E1 27526.691,E2 27526.691} C_VEL
LIN {X 0,Y 583.128,Z 442.854,A -85,B 0,C 180,E1 27525.936,E2 27525.936} C_VEL
LIN {X 0,Y 576.665,Z 443.653,A -85,B 0,C 180,E1 27523.815,E2 27523.815} C_VEL
LIN {X 0,Y 576.154,Z 443.72,A -85,B 0,C 180,E1 27523.263,E2 27523.263} C_VEL
LIN {X 0,Y 576.16,Z 443.718,A -85,B 0,C 180,E1 27520.009,E2 27520.009} C_VEL
LIN {X 0,Y 576.144,Z 443.718,A -85,B 0,C 180,E1 27516.692,E2 27516.692} C_VEL
LIN {X 0,Y 576.158,Z 443.719,A -85,B 0,C 180,E1 27513.344,E2 27513.344} C_VEL
LIN {X 0,Y 576.16,Z 443.72,A -85,B 0,C 180,E1 27509.991,E2 27509.991} C_VEL
LIN {X 0,Y 576.157,Z 443.721,A -85,B 0,C 180,E1 27506.625,E2 27506.625} C_VEL
LIN {X 0,Y 576.159,Z 443.721,A -85,B 0,C 180,E1 27503.297,E2 27503.297} C_VEL
LIN {X 0,Y 576.162,Z 443.718,A -85,B 0,C 180,E1 27499.922,E2 27499.922} C_VEL
LIN {X 0,Y 576.156,Z 443.719,A -85,B 0,C 180,E1 27496.59,E2 27496.59} C_VEL
LIN {X 0,Y 576.15,Z 443.723,A -85,B 0,C 180,E1 27493.273,E2 27493.273} C_VEL
LIN {X 0,Y 576.157,Z 443.72,A -85,B 0,C 180,E1 27490.065,E2 27490.065} C_VEL
LIN {X 0,Y 576.159,Z 443.721,A -85,B 0,C 180,E1 27486.702,E2 27486.702} C_VEL
LIN {X 0,Y 576.162,Z 443.718,A -85,B 0,C 180,E1 27483.315,E2 27483.315} C_VEL
LIN {X 0,Y 576.217,Z 444.089,A -85,B 0,C 180,E1 27483.241,E2 27483.241} C_VEL
LIN {X 0,Y 579.162,Z 452.946,A -85,B 0,C 180,E1 27482.356,E2 27482.356} C_VEL
LIN {X 0,Y 578.569,Z 495.028,A -85,B 0,C 180,E1 27479.165,E2 27479.165} C_VEL
LIN {X 0,Y 579.681,Z 501.992,A -85,B 0,C 180,E1 27479.007,E2 27479.007} C_VEL
LIN {X 0,Y 578.896,Z 742.783,A -85,B 0,C 180,E1 27475.753,E2 27475.753} C_VEL
LIN {X 0,Y 578.756,Z 764.935,A -85,B 0,C 180,E1 27475.371,E2 27475.371} C_VEL
LIN {X 0,Y 578.512,Z 785.824,A -85,B 0,C 180,E1 27474.816,E2 27474.816} C_VEL
LIN {X 0,Y 578.225,Z 806.191,A -85,B 0,C 180,E1 27474.075,E2 27474.075} C_VEL
LIN {X 0,Y 577.923,Z 825.48,A -85,B 0,C 180,E1 27473.178,E2 27473.178} C_VEL
LIN {X 0,Y 577.624,Z 844.064,A -85,B 0,C 180,E1 27472.116,E2 27472.116} C_VEL
LIN {X 0,Y 577.287,Z 861.649,A -85,B 0,C 180,E1 27470.903,E2 27470.903} C_VEL
LIN {X 0,Y 576.966,Z 878.329,A -85,B 0,C 180,E1 27469.539,E2 27469.539} C_VEL
LIN {X 0,Y 576.687,Z 894.03,A -85,B 0,C 180,E1 27468.029,E2 27468.029} C_VEL
LIN {X 0,Y 576.449,Z 908.245,A -85,B 0,C 180,E1 27466.422,E2 27466.422} C_VEL
LIN {X 0,Y 576.265,Z 921.386,A -85,B 0,C 180,E1 27464.674,E2 27464.674} C_VEL
LIN {X 0,Y 576.124,Z 933.014,A -85,B 0,C 180,E1 27462.834,E2 27462.834} C_VEL
LIN {X 0,Y 576.024,Z 942.674,A -85,B 0,C 180,E1 27461.007,E2 27461.007} C_VEL
LIN {X 0,Y 575.957,Z 950.912,A -85,B 0,C 180,E1 27459.089,E2 27459.089} C_VEL
LIN {X 0,Y 575.92,Z 957.374,A -85,B 0,C 180,E1 27457.18,E2 27457.18} C_VEL
LIN {X 0,Y 575.905,Z 962.462,A -85,B 0,C 180,E1 27455.179,E2 27455.179} C_VEL
LIN {X 0,Y 575.9,Z 965.893,A -85,B 0,C 180,E1 27453.184,E2 27453.184} C_VEL
LIN {X 0,Y 575.902,Z 967.676,A -85,B 0,C 180,E1 27451.193,E2 27451.193} C_VEL
LIN {X 0,Y 575.906,Z 967.839,A -85,B 0,C 180,E1 27449.204,E2 27449.204} C_VEL
LIN {X 0,Y 575.911,Z 966.442,A -85,B 0,C 180,E1 27447.213,E2 27447.213} C_VEL
LIN {X 0,Y 575.919,Z 963.464,A -85,B 0,C 180,E1 27445.219,E2 27445.219} C_VEL
LIN {X 0,Y 575.932,Z 958.833,A -85,B 0,C 180,E1 27443.22,E2 27443.22} C_VEL
LIN {X 0,Y 575.957,Z 952.364,A -85,B 0,C 180,E1 27441.212,E2 27441.212} C_VEL
LIN {X 0,Y 576.004,Z 944.319,A -85,B 0,C 180,E1 27439.264,E2 27439.264} C_VEL
LIN {X 0,Y 576.105,Z 934.673,A -85,B 0,C 180,E1 27437.368,E2 27437.368} C_VEL
LIN {X 0,Y 576.238,Z 923.307,A -85,B 0,C 180,E1 27435.516,E2 27435.516} C_VEL
LIN {X 0,Y 576.424,Z 910.65,A -85,B 0,C 180,E1 27433.783,E2 27433.783} C_VEL
LIN {X 0,Y 576.658,Z 896.4,A -85,B 0,C 180,E1 27432.127,E2 27432.127} C_VEL
LIN {X 0,Y 576.946,Z 880.536,A -85,B 0,C 180,E1 27430.564,E2 27430.564} C_VEL
LIN {X 0,Y 577.252,Z 863.82,A -85,B 0,C 180,E1 27429.171,E2 27429.171} C_VEL
LIN {X 0,Y 577.567,Z 846.207,A -85,B 0,C 180,E1 27427.934,E2 27427.934} C_VEL
LIN {X 0,Y 577.863,Z 828.116,A -85,B 0,C 180,E1 27426.872,E2 27426.872} C_VEL
LIN {X 0,Y 578.201,Z 808.056,A -85,B 0,C 180,E1 27425.914,E2 27425.914} C_VEL
LIN {X 0,Y 578.501,Z 787.401,A -85,B 0,C 180,E1 27425.144,E2 27425.144} C_VEL
LIN {X 0,Y 578.736,Z 766.739,A -85,B 0,C 180,E1 27424.578,E2 27424.578} C_VEL
LIN {X 0,Y 578.889,Z 745.786,A -85,B 0,C 180,E1 27424.198,E2 27424.198} C_VEL
LIN {X 0,Y 579.609,Z 504.494,A -85,B 0,C 180,E1 27420.934,E2 27420.934} C_VEL
LIN {X 0,Y 577.81,Z 497.279,A -85,B 0,C 180,E1 27420.708,E2 27420.708} C_VEL
LIN {X 0,Y 578.209,Z 469.525,A -85,B 0,C 180,E1 27417.551,E2 27417.551} C_VEL
LIN {X 0,Y 578.459,Z 451.664,A -85,B 0,C 180,E1 27415.462,E2 27415.462} C_VEL
LIN {X 0,Y 576.115,Z 443.72,A -85,B 0,C 180,E1 27414.314,E2 27414.314} C_VEL
LIN {X 0,Y 576.163,Z 443.722,A -85,B 0,C 180,E1 27411.186,E2 27411.186} C_VEL
LIN {X 0,Y 576.121,Z 443.718,A -85,B 0,C 180,E1 27407.94,E2 27407.94} C_VEL
LIN {X 0,Y 576.154,Z 443.714,A -85,B 0,C 180,E1 27404.782,E2 27404.782} C_VEL
LIN {X 0,Y 576.141,Z 443.718,A -85,B 0,C 180,E1 27401.525,E2 27401.525} C_VEL
LIN {X 0,Y 576.155,Z 443.712,A -85,B 0,C 180,E1 27398.156,E2 27398.156} C_VEL
LIN {X 0,Y 576.141,Z 443.719,A -85,B 0,C 180,E1 27394.817,E2 27394.817} C_VEL
LIN {X 0,Y 576.149,Z 443.72,A -85,B 0,C 180,E1 27391.559,E2 27391.559} C_VEL
LIN {X 0,Y 576.132,Z 443.72,A -85,B 0,C 180,E1 27388.371,E2 27388.371} C_VEL
LIN {X 0,Y 576.178,Z 443.941,A -85,B 0,C 180,E1 27388.109,E2 27388.109} C_VEL
LIN {X 0,Y 578.702,Z 452.461,A -85,B 0,C 180,E1 27387.138,E2 27387.138} C_VEL
LIN {X 0,Y 578.32,Z 484.109,A -85,B 0,C 180,E1 27384.189,E2 27384.189} C_VEL
LIN {X 0,Y 577.682,Z 517.274,A -85,B 0,C 180,E1 27381.154,E2 27381.154} C_VEL
LIN {X 0,Y 577.087,Z 553.032,A -85,B 0,C 180,E1 27377.911,E2 27377.911} C_VEL
LIN {X 0,Y 576.779,Z 589.398,A -85,B 0,C 180,E1 27374.764,E2 27374.764} C_VEL
LIN {X 0,Y 576.7,Z 602.566,A -85,B 0,C 180,E1 27373.657,E2 27373.657} C_VEL
LIN {X 0,Y 577.135,Z 609.493,A -85,B 0,C 180,E1 27373.556,E2 27373.556} C_VEL
LIN {X 0,Y 576.883,Z 743.675,A -85,B 0,C 180,E1 27371.836,E2 27371.836} C_VEL
LIN {X 0,Y 576.798,Z 760.034,A -85,B 0,C 180,E1 27371.448,E2 27371.448} C_VEL
LIN {X 0,Y 576.677,Z 775.248,A -85,B 0,C 180,E1 27370.894,E2 27370.894} C_VEL
LIN {X 0,Y 576.55,Z 789.788,A -85,B 0,C 180,E1 27370.189,E2 27370.189} C_VEL
LIN {X 0,Y 576.395,Z 804.06,A -85,B 0,C 180,E1 27369.284,E2 27369.284} C_VEL
LIN {X 0,Y 576.27,Z 816.064,A -85,B 0,C 180,E1 27368.33,E2 27368.33} C_VEL
LIN {X 0,Y 576.154,Z 827.908,A -85,B 0,C 180,E1 27367.178,E2 27367.178} C_VEL
LIN {X 0,Y 576.054,Z 838.547,A -85,B 0,C 180,E1 27365.878,E2 27365.878} C_VEL
LIN {X 0,Y 575.991,Z 847.11,A -85,B 0,C 180,E1 27364.58,E2 27364.58} C_VEL
LIN {X 0,Y 575.944,Z 855.28,A -85,B 0,C 180,E1 27362.986,E2 27362.986} C_VEL
LIN {X 0,Y 575.924,Z 860.89,A -85,B 0,C 180,E1 27361.492,E2 27361.492} C_VEL
LIN {X 0,Y 575.918,Z 865.044,A -85,B 0,C 180,E1 27359.901,E2 27359.901} C_VEL
LIN {X 0,Y 575.913,Z 867.345,A -85,B 0,C 180,E1 27358.309,E2 27358.309} C_VEL
LIN {X 0,Y 575.915,Z 867.954,A -85,B 0,C 180,E1 27356.716,E2 27356.716} C_VEL
LIN {X 0,Y 575.914,Z 866.728,A -85,B 0,C 180,E1 27355.02,E2 27355.02} C_VEL
LIN {X 0,Y 575.918,Z 863.941,A -85,B 0,C 180,E1 27353.521,E2 27353.521} C_VEL
LIN {X 0,Y 575.928,Z 859.575,A -85,B 0,C 180,E1 27352.017,E2 27352.017} C_VEL
LIN {X 0,Y 575.959,Z 852.874,A -85,B 0,C 180,E1 27350.407,E2 27350.407} C_VEL
LIN {X 0,Y 575.998,Z 845.672,A -85,B 0,C 180,E1 27349.093,E2 27349.093} C_VEL
LIN {X 0,Y 576.074,Z 836.354,A -85,B 0,C 180,E1 27347.735,E2 27347.735} C_VEL
LIN {X 0,Y 576.176,Z 825.215,A -85,B 0,C 180,E1 27346.452,E2 27346.452} C_VEL
LIN {X 0,Y 576.293,Z 813.745,A -85,B 0,C 180,E1 27345.378,E2 27345.378} C_VEL
LIN {X 0,Y 576.438,Z 800.127,A -85,B 0,C 180,E1 27344.352,E2 27344.352} C_VEL
LIN {X 0,Y 576.568,Z 786.251,A -85,B 0,C 180,E1 27343.536,E2 27343.536} C_VEL
LIN {X 0,Y 576.721,Z 771.495,A -85,B 0,C 180,E1 27342.859,E2 27342.859} C_VEL
LIN {X 0,Y 576.814,Z 755.269,A -85,B 0,C 180,E1 27342.332,E2 27342.332} C_VEL
LIN {X 0,Y 576.892,Z 740.521,A -85,B 0,C 180,E1 27342.021,E2 27342.021} C_VEL
LIN {X 0,Y 576.919,Z 604.212,A -85,B 0,C 180,E1 27340.28,E2 27340.28} C_VEL
LIN {X 0,Y 576.66,Z 602.172,A -85,B 0,C 180,E1 27340.239,E2 27340.239} C_VEL
LIN {X 0,Y 576.97,Z 562.635,A -85,B 0,C 180,E1 27336.835,E2 27336.835} C_VEL
LIN {X 0,Y 578.376,Z 529.504,A -85,B 0,C 180,E1 27333.623,E2 27333.623} C_VEL
LIN {X 0,Y 580.518,Z 495.287,A -85,B 0,C 180,E1 27330.148,E2 27330.148} C_VEL
LIN {X 0,Y 581.888,Z 477.784,A -85,B 0,C 180,E1 27328.274,E2 27328.274} C_VEL
LIN {X 0,Y 582.848,Z 458.783,A -85,B 0,C 180,E1 27325.997,E2 27325.997} C_VEL
LIN {X 0,Y 580.404,Z 452.666,A -85,B 0,C 180,E1 27324.743,E2 27324.743} C_VEL
LIN {X 0,Y 578.71,Z 449.319,A -85,B 0,C 180,E1 27323.903,E2 27323.903} C_VEL
LIN {X 0,Y 578.065,Z 447.994,A -85,B 0,C 180,E1 27323.543,E2 27323.543} C_VEL
LIN {X 0,Y 576.204,Z 444.178,A -85,B 0,C 180,E1 27322.306,E2 27322.306} C_VEL
LIN {X 0,Y 576.138,Z 443.72,A -85,B 0,C 180,E1 27322.096,E2 27322.096} C_VEL
LIN {X 0,Y 576.134,Z 443.723,A -85,B 0,C 180,E1 27318.717,E2 27318.717} C_VEL
LIN {X 0,Y 576.159,Z 443.98,A -85,B 0,C 180,E1 27318.115,E2 27318.115} C_VEL
LIN {X 0,Y 577.739,Z 447.584,A -85,B 0,C 180,E1 27317.281,E2 27317.281} C_VEL
LIN {X 0,Y 578.685,Z 449.158,A -85,B 0,C 180,E1 27316.96,E2 27316.96} C_VEL
LIN {X 0,Y 581.331,Z 455.214,A -85,B 0,C 180,E1 27316.053,E2 27316.053} C_VEL
LIN {X 0,Y 579.808,Z 478.931,A -85,B 0,C 180,E1 27314.369,E2 27314.369} C_VEL
LIN {X 0,Y 578.642,Z 516.29,A -85,B 0,C 180,E1 27312.011,E2 27312.011} C_VEL
LIN {X 0,Y 579.003,Z 540.26,A -85,B 0,C 180,E1 27310.552,E2 27310.552} C_VEL
LIN {X 0,Y 580.79,Z 554.919,A -85,B 0,C 180,E1 27309.611,E2 27309.611} C_VEL
LIN {X 0,Y 583.974,Z 566.007,A -85,B 0,C 180,E1 27308.828,E2 27308.828} C_VEL
LIN {X 0,Y 587.946,Z 573.542,A -85,B 0,C 180,E1 27308.217,E2 27308.217} C_VEL
LIN {X 0,Y 591.442,Z 577.715,A -85,B 0,C 180,E1 27307.705,E2 27307.705} C_VEL
LIN {X 0,Y 594.635,Z 580.115,A -85,B 0,C 180,E1 27307.132,E2 27307.132} C_VEL
LIN {X 0,Y 596.787,Z 580.763,A -85,B 0,C 180,E1 27306.616,E2 27306.616} C_VEL
LIN {X 0,Y 598.348,Z 579.988,A -85,B 0,C 180,E1 27306.023,E2 27306.023} C_VEL
LIN {X 0,Y 598.768,Z 577.835,A -85,B 0,C 180,E1 27305.465,E2 27305.465} C_VEL
LIN {X 0,Y 597.992,Z 574.309,A -85,B 0,C 180,E1 27304.952,E2 27304.952} C_VEL
LIN {X 0,Y 596.067,Z 569.655,A -85,B 0,C 180,E1 27304.54,E2 27304.54} C_VEL
LIN {X 0,Y 593.143,Z 561.973,A -85,B 0,C 180,E1 27304.127,E2 27304.127} C_VEL
LIN {X 0,Y 591.082,Z 552.901,A -85,B 0,C 180,E1 27303.831,E2 27303.831} C_VEL
LIN {X 0,Y 589.902,Z 542.129,A -85,B 0,C 180,E1 27303.66,E2 27303.66} C_VEL
LIN {X 0,Y 589.613,Z 530.887,A -85,B 0,C 180,E1 27303.618,E2 27303.618} C_VEL
LIN {X 0,Y 589.486,Z 481.289,A -85,B 0,C 180,E1 27303.599,E2 27303.599} C_VEL
LIN {X 0,Y 584.961,Z 492.214,A -85,B 0,C 180,E1 27302.926,E2 27302.926} C_VEL
LIN {X 0,Y 581.991,Z 497.108,A -85,B 0,C 180,E1 27302.472,E2 27302.472} C_VEL
LIN {X 0,Y 580.12,Z 498.434,A -85,B 0,C 180,E1 27302.18,E2 27302.18} C_VEL
LIN {X 0,Y 579.45,Z 498.362,A -85,B 0,C 180,E1 27302.061,E2 27302.061} C_VEL
LIN {X 0,Y 578.876,Z 544.231,A -85,B 0,C 180,E1 27299.204,E2 27299.204} C_VEL
LIN {X 0,Y 579.627,Z 550.717,A -85,B 0,C 180,E1 27299.073,E2 27299.073} C_VEL
LIN {X 0,Y 578.83,Z 806.431,A -85,B 0,C 180,E1 27295.588,E2 27295.588} C_VEL
LIN {X 0,Y 578.621,Z 827.576,A -85,B 0,C 180,E1 27295.106,E2 27295.106} C_VEL
LIN {X 0,Y 578.368,Z 847.556,A -85,B 0,C 180,E1 27294.459,E2 27294.459} C_VEL
LIN {X 0,Y 578.069,Z 866.625,A -85,B 0,C 180,E1 27293.659,E2 27293.659} C_VEL
LIN {X 0,Y 577.758,Z 885.976,A -85,B 0,C 180,E1 27292.648,E2 27292.648} C_VEL
LIN {X 0,Y 577.434,Z 904.269,A -85,B 0,C 180,E1 27291.483,E2 27291.483} C_VEL
LIN {X 0,Y 577.106,Z 921.546,A -85,B 0,C 180,E1 27290.169,E2 27290.169} C_VEL
LIN {X 0,Y 576.799,Z 938.353,A -85,B 0,C 180,E1 27288.653,E2 27288.653} C_VEL
LIN {X 0,Y 576.54,Z 953.423,A -85,B 0,C 180,E1 27287.043,E2 27287.043} C_VEL
LIN {X 0,Y 576.327,Z 967.369,A -85,B 0,C 180,E1 27285.29,E2 27285.29} C_VEL
LIN {X 0,Y 576.159,Z 979.013,A -85,B 0,C 180,E1 27283.55,E2 27283.55} C_VEL
LIN {X 0,Y 576.044,Z 989.849,A -85,B 0,C 180,E1 27281.616,E2 27281.616} C_VEL
LIN {X 0,Y 575.976,Z 998.668,A -85,B 0,C 180,E1 27279.695,E2 27279.695} C_VEL
LIN {X 0,Y 575.943,Z 1005.986,A -85,B 0,C 180,E1 27277.683,E2 27277.683} C_VEL
LIN {X 0,Y 575.92,Z 1011.496,A -85,B 0,C 180,E1 27275.68,E2 27275.68} C_VEL
LIN {X 0,Y 575.905,Z 1015.409,A -85,B 0,C 180,E1 27273.584,E2 27273.584} C_VEL
LIN {X 0,Y 575.901,Z 1017.448,A -85,B 0,C 180,E1 27271.592,E2 27271.592} C_VEL
LIN {X 0,Y 575.9,Z 1017.896,A -85,B 0,C 180,E1 27269.503,E2 27269.503} C_VEL
LIN {X 0,Y 575.907,Z 1016.74,A -85,B 0,C 180,E1 27267.513,E2 27267.513} C_VEL
LIN {X 0,Y 575.915,Z 1013.77,A -85,B 0,C 180,E1 27265.42,E2 27265.42} C_VEL
LIN {X 0,Y 575.932,Z 1009.224,A -85,B 0,C 180,E1 27263.421,E2 27263.421} C_VEL
LIN {X 0,Y 575.959,Z 1002.926,A -85,B 0,C 180,E1 27261.414,E2 27261.414} C_VEL
LIN {X 0,Y 576.006,Z 994.732,A -85,B 0,C 180,E1 27259.398,E2 27259.398} C_VEL
LIN {X 0,Y 576.103,Z 984.983,A -85,B 0,C 180,E1 27257.471,E2 27257.471} C_VEL
LIN {X 0,Y 576.225,Z 974.505,A -85,B 0,C 180,E1 27255.736,E2 27255.736} C_VEL
LIN {X 0,Y 576.413,Z 961.541,A -85,B 0,C 180,E1 27253.941,E2 27253.941} C_VEL
LIN {X 0,Y 576.649,Z 946.963,A -85,B 0,C 180,E1 27252.232,E2 27252.232} C_VEL
LIN {X 0,Y 576.93,Z 931.164,A -85,B 0,C 180,E1 27250.67,E2 27250.67} C_VEL
LIN {X 0,Y 577.231,Z 914.734,A -85,B 0,C 180,E1 27249.287,E2 27249.287} C_VEL
LIN {X 0,Y 577.544,Z 897.175,A -85,B 0,C 180,E1 27248.041,E2 27248.041} C_VEL
LIN {X 0,Y 577.861,Z 878.344,A -85,B 0,C 180,E1 27246.929,E2 27246.929} C_VEL
LIN {X 0,Y 578.205,Z 858.326,A -85,B 0,C 180,E1 27245.969,E2 27245.969} C_VEL
LIN {X 0,Y 578.497,Z 838.295,A -85,B 0,C 180,E1 27245.217,E2 27245.217} C_VEL
LIN {X 0,Y 578.724,Z 818.003,A -85,B 0,C 180,E1 27244.651,E2 27244.651} C_VEL
LIN {X 0,Y 578.876,Z 796.829,A -85,B 0,C 180,E1 27244.259,E2 27244.259} C_VEL
LIN {X 0,Y 579.628,Z 550.422,A -85,B 0,C 180,E1 27240.923,E2 27240.923} C_VEL
LIN {X 0,Y 578.823,Z 543.467,A -85,B 0,C 180,E1 27240.764,E2 27240.764} C_VEL
LIN {X 0,Y 579.515,Z 498.199,A -85,B 0,C 180,E1 27237.915,E2 27237.915} C_VEL
LIN {X 0,Y 580.647,Z 498.291,A -85,B 0,C 180,E1 27237.737,E2 27237.737} C_VEL
LIN {X 0,Y 582.926,Z 495.834,A -85,B 0,C 180,E1 27237.384,E2 27237.384} C_VEL
LIN {X 0,Y 586.455,Z 488.972,A -85,B 0,C 180,E1 27236.849,E2 27236.849} C_VEL
LIN {X 0,Y 589.549,Z 481.254,A -85,B 0,C 180,E1 27236.392,E2 27236.392} C_VEL
LIN {X 0,Y 589.774,Z 539.722,A -85,B 0,C 180,E1 27236.359,E2 27236.359} C_VEL
LIN {X 0,Y 590.78,Z 550.928,A -85,B 0,C 180,E1 27236.212,E2 27236.212} C_VEL
LIN {X 0,Y 592.646,Z 560.205,A -85,B 0,C 180,E1 27235.944,E2 27235.944} C_VEL
LIN {X 0,Y 595.284,Z 567.914,A -85,B 0,C 180,E1 27235.57,E2 27235.57} C_VEL
LIN {X 0,Y 597.588,Z 573.18,A -85,B 0,C 180,E1 27235.168,E2 27235.168} C_VEL
LIN {X 0,Y 598.667,Z 576.865,A -85,B 0,C 180,E1 27234.7,E2 27234.7} C_VEL
LIN {X 0,Y 598.675,Z 579.201,A -85,B 0,C 180,E1 27234.23,E2 27234.23} C_VEL
LIN {X 0,Y 597.717,Z 580.569,A -85,B 0,C 180,E1 27233.689,E2 27233.689} C_VEL
LIN {X 0,Y 595.936,Z 580.641,A -85,B 0,C 180,E1 27233.159,E2 27233.159} C_VEL
LIN {X 0,Y 593.062,Z 579.104,A -85,B 0,C 180,E1 27232.567,E2 27232.567} C_VEL
LIN {X 0,Y 589.731,Z 575.876,A -85,B 0,C 180,E1 27232.034,E2 27232.034} C_VEL
LIN {X 0,Y 585.932,Z 569.991,A -85,B 0,C 180,E1 27231.403,E2 27231.403} C_VEL
LIN {X 0,Y 583.039,Z 561.704,A -85,B 0,C 180,E1 27230.662,E2 27230.662} C_VEL
LIN {X 0,Y 581.213,Z 550.691,A -85,B 0,C 180,E1 27229.801,E2 27229.801} C_VEL
LIN {X 0,Y 580.617,Z 532.266,A -85,B 0,C 180,E1 27228.512,E2 27228.512} C_VEL
LIN {X 0,Y 581.341,Z 494.767,A -85,B 0,C 180,E1 27225.924,E2 27225.924} C_VEL
LIN {X 0,Y 582.08,Z 456.768,A -85,B 0,C 180,E1 27223.186,E2 27223.186} C_VEL
LIN {X 0,Y 577.69,Z 447.547,A -85,B 0,C 180,E1 27222.053,E2 27222.053} C_VEL
LIN {X 0,Y 576.226,Z 444.267,A -85,B 0,C 180,E1 27221.65,E2 27221.65} C_VEL
LIN {X 0,Y 576.141,Z 443.724,A -85,B 0,C 180,E1 27221.585,E2 27221.585} C_VEL
LIN {X 0,Y 576.157,Z 443.72,A -85,B 0,C 180,E1 27218.282,E2 27218.282} C_VEL
LIN {X 0,Y 576.128,Z 443.722,A -85,B 0,C 180,E1 27214.939,E2 27214.939} C_VEL
LIN {X 0,Y 576.153,Z 443.715,A -85,B 0,C 180,E1 27211.607,E2 27211.607} C_VEL
LIN {X 0,Y 576.11,Z 443.721,A -85,B 0,C 180,E1 27208.507,E2 27208.507} C_VEL
LIN {X 0,Y 576.134,Z 443.718,A -85,B 0,C 180,E1 27205.272,E2 27205.272} C_VEL
LIN {X 0,Y 576.136,Z 443.717,A -85,B 0,C 180,E1 27202.07,E2 27202.07} C_VEL
LIN {X 0,Y 576.106,Z 443.721,A -85,B 0,C 180,E1 27198.728,E2 27198.728} C_VEL
LIN {X 0,Y 576.16,Z 443.714,A -85,B 0,C 180,E1 27195.5,E2 27195.5} C_VEL
LIN {X 0,Y 576.104,Z 443.721,A -85,B 0,C 180,E1 27192.283,E2 27192.283} C_VEL
LIN {X 0,Y 576.134,Z 443.717,A -85,B 0,C 180,E1 27188.885,E2 27188.885} C_VEL
LIN {X 0,Y 576.13,Z 443.718,A -85,B 0,C 180,E1 27185.777,E2 27185.777} C_VEL
LIN {X 0,Y 576.103,Z 443.721,A -85,B 0,C 180,E1 27182.387,E2 27182.387} C_VEL
LIN {X 0,Y 576.151,Z 443.716,A -85,B 0,C 180,E1 27179.304,E2 27179.304} C_VEL
LIN {X 0,Y 576.115,Z 443.72,A -85,B 0,C 180,E1 27176.019,E2 27176.019} C_VEL
LIN {X 0,Y 576.157,Z 443.712,A -85,B 0,C 180,E1 27172.722,E2 27172.722} C_VEL
LIN {X 0,Y 576.134,Z 443.718,A -85,B 0,C 180,E1 27169.399,E2 27169.399} C_VEL
LIN {X 0,Y 576.121,Z 443.72,A -85,B 0,C 180,E1 27166.143,E2 27166.143} C_VEL
LIN {X 0,Y 576.154,Z 443.72,A -85,B 0,C 180,E1 27163.263,E2 27163.263} C_VEL
LIN {X 0,Y 575.211,Z 443.846,A -85,B 0,C 180,E1 27162.497,E2 27162.497} C_VEL
LIN {X 0,Y 568.682,Z 444.658,A -85,B 0,C 180,E1 27160.292,E2 27160.292} C_VEL
LIN {X 0,Y 568.208,Z 444.71,A -85,B 0,C 180,E1 27159.787,E2 27159.787} C_VEL
LIN {X 0,Y 568.222,Z 444.708,A -85,B 0,C 180,E1 27156.456,E2 27156.456} C_VEL
LIN {X 0,Y 568.212,Z 444.707,A -85,B 0,C 180,E1 27153.113,E2 27153.113} C_VEL
LIN {X 0,Y 568.204,Z 444.707,A -85,B 0,C 180,E1 27149.783,E2 27149.783} C_VEL
LIN {X 0,Y 568.22,Z 444.708,A -85,B 0,C 180,E1 27146.518,E2 27146.518} C_VEL
LIN {X 0,Y 568.211,Z 444.709,A -85,B 0,C 180,E1 27143.191,E2 27143.191} C_VEL
LIN {X 0,Y 568.225,Z 444.705,A -85,B 0,C 180,E1 27139.776,E2 27139.776} C_VEL
LIN {X 0,Y 568.21,Z 444.709,A -85,B 0,C 180,E1 27136.467,E2 27136.467} C_VEL
LIN {X 0,Y 568.203,Z 444.712,A -85,B 0,C 180,E1 27133.197,E2 27133.197} C_VEL
LIN {X 0,Y 568.218,Z 444.708,A -85,B 0,C 180,E1 27129.961,E2 27129.961} C_VEL
LIN {X 0,Y 568.213,Z 444.711,A -85,B 0,C 180,E1 27126.621,E2 27126.621} C_VEL
LIN {X 0,Y 568.185,Z 444.712,A -85,B 0,C 180,E1 27123.724,E2 27123.724} C_VEL
LIN {X 0,Y 571.994,Z 455.956,A -85,B 0,C 180,E1 27122.574,E2 27122.574} C_VEL
LIN {X 0,Y 571.359,Z 495.363,A -85,B 0,C 180,E1 27119.566,E2 27119.566} C_VEL
LIN {X 0,Y 572.683,Z 503.21,A -85,B 0,C 180,E1 27119.38,E2 27119.38} C_VEL
LIN {X 0,Y 571.686,Z 744.742,A -85,B 0,C 180,E1 27116.075,E2 27116.075} C_VEL
LIN {X 0,Y 571.501,Z 766.031,A -85,B 0,C 180,E1 27115.692,E2 27115.692} C_VEL
LIN {X 0,Y 571.198,Z 787.014,A -85,B 0,C 180,E1 27115.118,E2 27115.118} C_VEL
LIN {X 0,Y 570.836,Z 807.265,A -85,B 0,C 180,E1 27114.361,E2 27114.361} C_VEL
LIN {X 0,Y 570.422,Z 827.483,A -85,B 0,C 180,E1 27113.391,E2 27113.391} C_VEL
LIN {X 0,Y 570.043,Z 845.688,A -85,B 0,C 180,E1 27112.317,E2 27112.317} C_VEL
LIN {X 0,Y 569.641,Z 863.092,A -85,B 0,C 180,E1 27111.089,E2 27111.089} C_VEL
LIN {X 0,Y 569.232,Z 880.13,A -85,B 0,C 180,E1 27109.655,E2 27109.655} C_VEL
LIN {X 0,Y 568.877,Z 895.552,A -85,B 0,C 180,E1 27108.125,E2 27108.125} C_VEL
LIN {X 0,Y 568.576,Z 909.935,A -85,B 0,C 180,E1 27106.446,E2 27106.446} C_VEL
LIN {X 0,Y 568.337,Z 923.139,A -85,B 0,C 180,E1 27104.624,E2 27104.624} C_VEL
LIN {X 0,Y 568.159,Z 934.753,A -85,B 0,C 180,E1 27102.707,E2 27102.707} C_VEL
LIN {X 0,Y 568.033,Z 944.524,A -85,B 0,C 180,E1 27100.753,E2 27100.753} C_VEL
LIN {X 0,Y 567.967,Z 952.409,A -85,B 0,C 180,E1 27098.809,E2 27098.809} C_VEL
LIN {X 0,Y 567.937,Z 958.866,A -85,B 0,C 180,E1 27096.774,E2 27096.774} C_VEL
LIN {X 0,Y 567.918,Z 963.488,A -85,B 0,C 180,E1 27094.746,E2 27094.746} C_VEL
LIN {X 0,Y 567.913,Z 966.454,A -85,B 0,C 180,E1 27092.724,E2 27092.724} C_VEL
LIN {X 0,Y 567.904,Z 967.864,A -85,B 0,C 180,E1 27090.605,E2 27090.605} C_VEL
LIN {X 0,Y 567.899,Z 967.602,A -85,B 0,C 180,E1 27088.587,E2 27088.587} C_VEL
LIN {X 0,Y 567.901,Z 965.767,A -85,B 0,C 180,E1 27086.568,E2 27086.568} C_VEL
LIN {X 0,Y 567.908,Z 962.233,A -85,B 0,C 180,E1 27084.544,E2 27084.544} C_VEL
LIN {X 0,Y 567.933,Z 957.034,A -85,B 0,C 180,E1 27082.514,E2 27082.514} C_VEL
LIN {X 0,Y 567.986,Z 950.057,A -85,B 0,C 180,E1 27080.475,E2 27080.475} C_VEL
LIN {X 0,Y 568.076,Z 941.616,A -85,B 0,C 180,E1 27078.527,E2 27078.527} C_VEL
LIN {X 0,Y 568.213,Z 931.186,A -85,B 0,C 180,E1 27076.568,E2 27076.568} C_VEL
LIN {X 0,Y 568.413,Z 919.169,A -85,B 0,C 180,E1 27074.7,E2 27074.7} C_VEL
LIN {X 0,Y 568.677,Z 905.575,A -85,B 0,C 180,E1 27072.924,E2 27072.924} C_VEL
LIN {X 0,Y 568.988,Z 890.833,A -85,B 0,C 180,E1 27071.292,E2 27071.292} C_VEL
LIN {X 0,Y 569.341,Z 875.391,A -85,B 0,C 180,E1 27069.836,E2 27069.836} C_VEL
LIN {X 0,Y 569.737,Z 858.139,A -85,B 0,C 180,E1 27068.454,E2 27068.454} C_VEL
LIN {X 0,Y 570.169,Z 839.358,A -85,B 0,C 180,E1 27067.197,E2 27067.197} C_VEL
LIN {X 0,Y 570.594,Z 819.763,A -85,B 0,C 180,E1 27066.122,E2 27066.122} C_VEL
LIN {X 0,Y 570.988,Z 800.131,A -85,B 0,C 180,E1 27065.259,E2 27065.259} C_VEL
LIN {X 0,Y 571.318,Z 779.821,A -85,B 0,C 180,E1 27064.57,E2 27064.57} C_VEL
LIN {X 0,Y 571.572,Z 758.925,A -85,B 0,C 180,E1 27064.066,E2 27064.066} C_VEL
LIN {X 0,Y 571.768,Z 724.418,A -85,B 0,C 180,E1 27063.56,E2 27063.56} C_VEL
LIN {X 0,Y 572.574,Z 505.93,A -85,B 0,C 180,E1 27060.563,E2 27060.563} C_VEL
LIN {X 0,Y 570.373,Z 497.352,A -85,B 0,C 180,E1 27060.297,E2 27060.297} C_VEL
LIN {X 0,Y 570.834,Z 470.71,A -85,B 0,C 180,E1 27057.22,E2 27057.22} C_VEL
LIN {X 0,Y 571.172,Z 454.68,A -85,B 0,C 180,E1 27055.324,E2 27055.324} C_VEL
LIN {X 0,Y 568.171,Z 444.712,A -85,B 0,C 180,E1 27053.907,E2 27053.907} C_VEL
LIN {X 0,Y 568.212,Z 444.706,A -85,B 0,C 180,E1 27050.578,E2 27050.578} C_VEL
LIN {X 0,Y 568.219,Z 444.71,A -85,B 0,C 180,E1 27047.217,E2 27047.217} C_VEL
LIN {X 0,Y 568.19,Z 444.704,A -85,B 0,C 180,E1 27043.895,E2 27043.895} C_VEL
LIN {X 0,Y 568.212,Z 444.703,A -85,B 0,C 180,E1 27040.623,E2 27040.623} C_VEL
LIN {X 0,Y 568.216,Z 444.71,A -85,B 0,C 180,E1 27037.252,E2 27037.252} C_VEL
LIN {X 0,Y 568.21,Z 444.705,A -85,B 0,C 180,E1 27033.843,E2 27033.843} C_VEL
LIN {X 0,Y 568.196,Z 444.71,A -85,B 0,C 180,E1 27030.568,E2 27030.568} C_VEL
LIN {X 0,Y 568.226,Z 444.957,A -85,B 0,C 180,E1 27028.538,E2 27028.538} C_VEL
LIN {X 0,Y 571.444,Z 455.204,A -85,B 0,C 180,E1 27027.342,E2 27027.342} C_VEL
LIN {X 0,Y 570.983,Z 486.424,A -85,B 0,C 180,E1 27024.41,E2 27024.41} C_VEL
LIN {X 0,Y 570.26,Z 519.739,A -85,B 0,C 180,E1 27021.335,E2 27021.335} C_VEL
LIN {X 0,Y 569.568,Z 556.301,A -85,B 0,C 180,E1 27017.997,E2 27017.997} C_VEL
LIN {X 0,Y 569.008,Z 589.916,A -85,B 0,C 180,E1 27014.97,E2 27014.97} C_VEL
LIN {X 0,Y 568.938,Z 602.725,A -85,B 0,C 180,E1 27013.89,E2 27013.89} C_VEL
LIN {X 0,Y 569.468,Z 609.646,A -85,B 0,C 180,E1 27013.784,E2 27013.784} C_VEL
LIN {X 0,Y 569.146,Z 743.334,A -85,B 0,C 180,E1 27012.048,E2 27012.048} C_VEL
LIN {X 0,Y 569.039,Z 759.795,A -85,B 0,C 180,E1 27011.658,E2 27011.658} C_VEL
LIN {X 0,Y 568.903,Z 773.858,A -85,B 0,C 180,E1 27011.147,E2 27011.147} C_VEL
LIN {X 0,Y 568.741,Z 786.739,A -85,B 0,C 180,E1 27010.535,E2 27010.535} C_VEL
LIN {X 0,Y 568.585,Z 800.355,A -85,B 0,C 180,E1 27009.719,E2 27009.719} C_VEL
LIN {X 0,Y 568.392,Z 814.232,A -85,B 0,C 180,E1 27008.65,E2 27008.65} C_VEL
LIN {X 0,Y 568.246,Z 825.427,A -85,B 0,C 180,E1 27007.583,E2 27007.583} C_VEL
LIN {X 0,Y 568.116,Z 836.664,A -85,B 0,C 180,E1 27006.265,E2 27006.265} C_VEL
LIN {X 0,Y 568.023,Z 845.672,A -85,B 0,C 180,E1 27004.925,E2 27004.925} C_VEL
LIN {X 0,Y 567.968,Z 853.18,A -85,B 0,C 180,E1 27003.533,E2 27003.533} C_VEL
LIN {X 0,Y 567.93,Z 859.724,A -85,B 0,C 180,E1 27001.917,E2 27001.917} C_VEL
LIN {X 0,Y 567.918,Z 864.012,A -85,B 0,C 180,E1 27000.404,E2 27000.404} C_VEL
LIN {X 0,Y 567.916,Z 866.891,A -85,B 0,C 180,E1 26998.79,E2 26998.79} C_VEL
LIN {X 0,Y 567.915,Z 867.944,A -85,B 0,C 180,E1 26997.074,E2 26997.074} C_VEL
LIN {X 0,Y 567.913,Z 867.316,A -85,B 0,C 180,E1 26995.557,E2 26995.557} C_VEL
LIN {X 0,Y 567.917,Z 864.779,A -85,B 0,C 180,E1 26993.835,E2 26993.835} C_VEL
LIN {X 0,Y 567.93,Z 860.742,A -85,B 0,C 180,E1 26992.311,E2 26992.311} C_VEL
LIN {X 0,Y 567.953,Z 855.451,A -85,B 0,C 180,E1 26990.884,E2 26990.884} C_VEL
LIN {X 0,Y 568.01,Z 847.243,A -85,B 0,C 180,E1 26989.246,E2 26989.246} C_VEL
LIN {X 0,Y 568.085,Z 839.296,A -85,B 0,C 180,E1 26988.013,E2 26988.013} C_VEL
LIN {X 0,Y 568.199,Z 829.572,A -85,B 0,C 180,E1 26986.776,E2 26986.776} C_VEL
LIN {X 0,Y 568.357,Z 817.026,A -85,B 0,C 180,E1 26985.506,E2 26985.506} C_VEL
LIN {X 0,Y 568.511,Z 805.142,A -85,B 0,C 180,E1 26984.535,E2 26984.535} C_VEL
LIN {X 0,Y 568.708,Z 791.097,A -85,B 0,C 180,E1 26983.61,E2 26983.61} C_VEL
LIN {X 0,Y 568.869,Z 776.541,A -85,B 0,C 180,E1 26982.878,E2 26982.878} C_VEL
LIN {X 0,Y 568.998,Z 762.868,A -85,B 0,C 180,E1 26982.355,E2 26982.355} C_VEL
LIN {X 0,Y 569.134,Z 746.563,A -85,B 0,C 180,E1 26981.918,E2 26981.918} C_VEL
LIN {X 0,Y 569.237,Z 719.426,A -85,B 0,C 180,E1 26981.531,E2 26981.531} C_VEL
LIN {X 0,Y 569.235,Z 604.919,A -85,B 0,C 180,E1 26980.058,E2 26980.058} C_VEL
LIN {X 0,Y 568.876,Z 602.257,A -85,B 0,C 180,E1 26980.01,E2 26980.01} C_VEL
LIN {X 0,Y 569.121,Z 584.881,A -85,B 0,C 180,E1 26978.458,E2 26978.458} C_VEL
LIN {X 0,Y 570.633,Z 549.461,A -85,B 0,C 180,E1 26975.022,E2 26975.022} C_VEL
LIN {X 0,Y 572.646,Z 515.408,A -85,B 0,C 180,E1 26971.589,E2 26971.589} C_VEL
LIN {X 0,Y 575.395,Z 484.311,A -85,B 0,C 180,E1 26968.288,E2 26968.288} C_VEL
LIN {X 0,Y 576.812,Z 463.668,A -85,B 0,C 180,E1 26965.777,E2 26965.777} C_VEL
LIN {X 0,Y 574.332,Z 457.65,A -85,B 0,C 180,E1 26964.447,E2 26964.447} C_VEL
LIN {X 0,Y 572.669,Z 453.84,A -85,B 0,C 180,E1 26963.432,E2 26963.432} C_VEL
LIN {X 0,Y 571.03,Z 450.097,A -85,B 0,C 180,E1 26962.157,E2 26962.157} C_VEL
LIN {X 0,Y 569.572,Z 448.284,A -85,B 0,C 180,E1 26960.729,E2 26960.729} C_VEL
LIN {X 0,Y 569.542,Z 448.209,A -85,B 0,C 180,E1 26959.624,E2 26959.624} C_VEL
LIN {X 0,Y 570.661,Z 449.569,A -85,B 0,C 180,E1 26958.525,E2 26958.525} C_VEL
LIN {X 0,Y 571.235,Z 450.478,A -85,B 0,C 180,E1 26958.173,E2 26958.173} C_VEL
LIN {X 0,Y 572.923,Z 454.031,A -85,B 0,C 180,E1 26957.285,E2 26957.285} C_VEL
LIN {X 0,Y 575.136,Z 459.522,A -85,B 0,C 180,E1 26956.373,E2 26956.373} C_VEL
LIN {X 0,Y 573.184,Z 480.955,A -85,B 0,C 180,E1 26954.768,E2 26954.768} C_VEL
LIN {X 0,Y 571.638,Z 514.078,A -85,B 0,C 180,E1 26952.577,E2 26952.577} C_VEL
LIN {X 0,Y 571.585,Z 540.548,A -85,B 0,C 180,E1 26950.915,E2 26950.915} C_VEL
LIN {X 0,Y 573.267,Z 556.415,A -85,B 0,C 180,E1 26949.877,E2 26949.877} C_VEL
LIN {X 0,Y 576.272,Z 567.89,A -85,B 0,C 180,E1 26949.065,E2 26949.065} C_VEL
LIN {X 0,Y 580.352,Z 576.53,A -85,B 0,C 180,E1 26948.382,E2 26948.382} C_VEL
LIN {X 0,Y 585.57,Z 583.16,A -85,B 0,C 180,E1 26947.761,E2 26947.761} C_VEL
LIN {X 0,Y 589.307,Z 586.233,A -85,B 0,C 180,E1 26947.275,E2 26947.275} C_VEL
LIN {X 0,Y 592.557,Z 587.816,A -85,B 0,C 180,E1 26946.727,E2 26946.727} C_VEL
LIN {X 0,Y 594.968,Z 587.889,A -85,B 0,C 180,E1 26946.148,E2 26946.148} C_VEL
LIN {X 0,Y 596.296,Z 586.605,A -85,B 0,C 180,E1 26945.581,E2 26945.581} C_VEL
LIN {X 0,Y 596.471,Z 584.159,A -85,B 0,C 180,E1 26945.039,E2 26945.039} C_VEL
LIN {X 0,Y 595.368,Z 580.442,A -85,B 0,C 180,E1 26944.528,E2 26944.528} C_VEL
LIN {X 0,Y 592.897,Z 575.378,A -85,B 0,C 180,E1 26944.092,E2 26944.092} C_VEL
LIN {X 0,Y 589.59,Z 566.99,A -85,B 0,C 180,E1 26943.614,E2 26943.614} C_VEL
LIN {X 0,Y 587.248,Z 557.485,A -85,B 0,C 180,E1 26943.269,E2 26943.269} C_VEL
LIN {X 0,Y 585.778,Z 546.415,A -85,B 0,C 180,E1 26943.049,E2 26943.049} C_VEL
LIN {X 0,Y 585.225,Z 533.408,A -85,B 0,C 180,E1 26942.966,E2 26942.966} C_VEL
LIN {X 0,Y 585.165,Z 502.758,A -85,B 0,C 180,E1 26942.957,E2 26942.957} C_VEL
LIN {X 0,Y 582.26,Z 505.728,A -85,B 0,C 180,E1 26942.513,E2 26942.513} C_VEL
LIN {X 0,Y 581.655,Z 506.9,A -85,B 0,C 180,E1 26942.42,E2 26942.42} C_VEL
LIN {X 0,Y 577.67,Z 517.205,A -85,B 0,C 180,E1 26941.792,E2 26941.792} C_VEL
LIN {X 0,Y 574.597,Z 522.738,A -85,B 0,C 180,E1 26941.294,E2 26941.294} C_VEL
LIN {X 0,Y 572.787,Z 524.327,A -85,B 0,C 180,E1 26940.995,E2 26940.995} C_VEL
LIN {X 0,Y 571.983,Z 524.19,A -85,B 0,C 180,E1 26940.854,E2 26940.854} C_VEL
LIN {X 0,Y 571.714,Z 544.425,A -85,B 0,C 180,E1 26939.604,E2 26939.604} C_VEL
LIN {X 0,Y 572.63,Z 551.734,A -85,B 0,C 180,E1 26939.448,E2 26939.448} C_VEL
LIN {X 0,Y 571.61,Z 806.417,A -85,B 0,C 180,E1 26935.935,E2 26935.935} C_VEL
LIN {X 0,Y 571.346,Z 827.68,A -85,B 0,C 180,E1 26935.445,E2 26935.445} C_VEL
LIN {X 0,Y 571.027,Z 847.569,A -85,B 0,C 180,E1 26934.795,E2 26934.795} C_VEL
LIN {X 0,Y 570.662,Z 866.632,A -85,B 0,C 180,E1 26933.985,E2 26933.985} C_VEL
LIN {X 0,Y 570.269,Z 885.89,A -85,B 0,C 180,E1 26932.968,E2 26932.968} C_VEL
LIN {X 0,Y 569.849,Z 904.27,A -85,B 0,C 180,E1 26931.784,E2 26931.784} C_VEL
LIN {X 0,Y 569.432,Z 921.542,A -85,B 0,C 180,E1 26930.453,E2 26930.453} C_VEL
LIN {X 0,Y 569.047,Z 938.347,A -85,B 0,C 180,E1 26928.916,E2 26928.916} C_VEL
LIN {X 0,Y 568.712,Z 953.419,A -85,B 0,C 180,E1 26927.285,E2 26927.285} C_VEL
LIN {X 0,Y 568.443,Z 967.363,A -85,B 0,C 180,E1 26925.508,E2 26925.508} C_VEL
LIN {X 0,Y 568.236,Z 979.014,A -85,B 0,C 180,E1 26923.742,E2 26923.742} C_VEL
LIN {X 0,Y 568.083,Z 989.852,A -85,B 0,C 180,E1 26921.781,E2 26921.781} C_VEL
LIN {X 0,Y 567.995,Z 998.672,A -85,B 0,C 180,E1 26919.832,E2 26919.832} C_VEL
LIN {X 0,Y 567.952,Z 1005.982,A -85,B 0,C 180,E1 26917.791,E2 26917.791} C_VEL
LIN {X 0,Y 567.925,Z 1011.494,A -85,B 0,C 180,E1 26915.76,E2 26915.76} C_VEL
LIN {X 0,Y 567.909,Z 1015.409,A -85,B 0,C 180,E1 26913.634,E2 26913.634} C_VEL
LIN {X 0,Y 567.902,Z 1017.45,A -85,B 0,C 180,E1 26911.615,E2 26911.615} C_VEL
LIN {X 0,Y 567.9,Z 1017.896,A -85,B 0,C 180,E1 26909.496,E2 26909.496} C_VEL
LIN {X 0,Y 567.907,Z 1016.744,A -85,B 0,C 180,E1 26907.478,E2 26907.478} C_VEL
LIN {X 0,Y 567.917,Z 1013.766,A -85,B 0,C 180,E1 26905.355,E2 26905.355} C_VEL
LIN {X 0,Y 567.934,Z 1009.476,A -85,B 0,C 180,E1 26903.43,E2 26903.43} C_VEL
LIN {X 0,Y 567.969,Z 1003.283,A -85,B 0,C 180,E1 26901.395,E2 26901.395} C_VEL
LIN {X 0,Y 568.029,Z 995.197,A -85,B 0,C 180,E1 26899.35,E2 26899.35} C_VEL
LIN {X 0,Y 568.151,Z 985.558,A -85,B 0,C 180,E1 26897.396,E2 26897.396} C_VEL
LIN {X 0,Y 568.302,Z 975.152,A -85,B 0,C 180,E1 26895.637,E2 26895.637} C_VEL
LIN {X 0,Y 568.548,Z 961.928,A -85,B 0,C 180,E1 26893.763,E2 26893.763} C_VEL
LIN {X 0,Y 568.831,Z 947.889,A -85,B 0,C 180,E1 26892.086,E2 26892.086} C_VEL
LIN {X 0,Y 569.186,Z 932.301,A -85,B 0,C 180,E1 26890.503,E2 26890.503} C_VEL
LIN {X 0,Y 569.581,Z 915.396,A -85,B 0,C 180,E1 26889.049,E2 26889.049} C_VEL
LIN {X 0,Y 570.001,Z 897.181,A -85,B 0,C 180,E1 26887.735,E2 26887.735} C_VEL
LIN {X 0,Y 570.402,Z 878.325,A -85,B 0,C 180,E1 26886.608,E2 26886.608} C_VEL
LIN {X 0,Y 570.822,Z 858.338,A -85,B 0,C 180,E1 26885.638,E2 26885.638} C_VEL
LIN {X 0,Y 571.191,Z 838.085,A -85,B 0,C 180,E1 26884.872,E2 26884.872} C_VEL
LIN {X 0,Y 571.482,Z 817.695,A -85,B 0,C 180,E1 26884.299,E2 26884.299} C_VEL
LIN {X 0,Y 571.673,Z 796.496,A -85,B 0,C 180,E1 26883.905,E2 26883.905} C_VEL
LIN {X 0,Y 572.635,Z 550.547,A -85,B 0,C 180,E1 26880.535,E2 26880.535} C_VEL
LIN {X 0,Y 571.629,Z 543.788,A -85,B 0,C 180,E1 26880.38,E2 26880.38} C_VEL
LIN {X 0,Y 572.01,Z 524.103,A -85,B 0,C 180,E1 26879.135,E2 26879.135} C_VEL
LIN {X 0,Y 573.298,Z 524.081,A -85,B 0,C 180,E1 26878.92,E2 26878.92} C_VEL
LIN {X 0,Y 575.632,Z 521.171,A -85,B 0,C 180,E1 26878.537,E2 26878.537} C_VEL
LIN {X 0,Y 579.184,Z 513.657,A -85,B 0,C 180,E1 26877.967,E2 26877.967} C_VEL
LIN {X 0,Y 581.985,Z 505.906,A -85,B 0,C 180,E1 26877.529,E2 26877.529} C_VEL
LIN {X 0,Y 584.82,Z 503.222,A -85,B 0,C 180,E1 26877.095,E2 26877.095} C_VEL
LIN {X 0,Y 585.219,Z 502.682,A -85,B 0,C 180,E1 26877.035,E2 26877.035} C_VEL
LIN {X 0,Y 585.39,Z 540.248,A -85,B 0,C 180,E1 26877.009,E2 26877.009} C_VEL
LIN {X 0,Y 586.421,Z 552.309,A -85,B 0,C 180,E1 26876.854,E2 26876.854} C_VEL
LIN {X 0,Y 588.342,Z 562.529,A -85,B 0,C 180,E1 26876.569,E2 26876.569} C_VEL
LIN {X 0,Y 591.075,Z 571.195,A -85,B 0,C 180,E1 26876.17,E2 26876.17} C_VEL
LIN {X 0,Y 594.48,Z 578.475,A -85,B 0,C 180,E1 26875.667,E2 26875.667} C_VEL
LIN {X 0,Y 596.135,Z 582.6,A -85,B 0,C 180,E1 26875.203,E2 26875.203} C_VEL
LIN {X 0,Y 596.516,Z 585.648,A -85,B 0,C 180,E1 26874.671,E2 26874.671} C_VEL
LIN {X 0,Y 595.801,Z 587.368,A -85,B 0,C 180,E1 26874.149,E2 26874.149} C_VEL
LIN {X 0,Y 593.957,Z 588.028,A -85,B 0,C 180,E1 26873.577,E2 26873.577} C_VEL
LIN {X 0,Y 590.998,Z 587.214,A -85,B 0,C 180,E1 26872.99,E2 26872.99} C_VEL
LIN {X 0,Y 587.27,Z 584.71,A -85,B 0,C 180,E1 26872.446,E2 26872.446} C_VEL
LIN {X 0,Y 582.041,Z 578.917,A -85,B 0,C 180,E1 26871.726,E2 26871.726} C_VEL
LIN {X 0,Y 578.283,Z 571.721,A -85,B 0,C 180,E1 26870.998,E2 26870.998} C_VEL
LIN {X 0,Y 575.477,Z 561.618,A -85,B 0,C 180,E1 26870.126,E2 26870.126} C_VEL
LIN {X 0,Y 574.006,Z 547.872,A -85,B 0,C 180,E1 26869.085,E2 26869.085} C_VEL
LIN {X 0,Y 574.792,Z 495.529,A -85,B 0,C 180,E1 26865.422,E2 26865.422} C_VEL
LIN {X 0,Y 575.601,Z 460.71,A -85,B 0,C 180,E1 26862.875,E2 26862.875} C_VEL
LIN {X 0,Y 569.507,Z 448.171,A -85,B 0,C 180,E1 26861.287,E2 26861.287} C_VEL
LIN {X 0,Y 568.21,Z 444.712,A -85,B 0,C 180,E1 26860.855,E2 26860.855} C_VEL
LIN {X 0,Y 568.177,Z 444.71,A -85,B 0,C 180,E1 26857.508,E2 26857.508} C_VEL
LIN {X 0,Y 568.223,Z 444.705,A -85,B 0,C 180,E1 26854.207,E2 26854.207} C_VEL
LIN {X 0,Y 568.195,Z 444.709,A -85,B 0,C 180,E1 26850.919,E2 26850.919} C_VEL
LIN {X 0,Y 568.195,Z 444.709,A -85,B 0,C 180,E1 26847.682,E2 26847.682} C_VEL
